// TwinCAT 3 PLC project PMPS_Prototype_Arbiter
// Title: PMPS
// Company: SLAC
// ProjectVersion: 0.0.0
// ProgramVersion: 3.1.4022.1
// libraries:
//   LCLS General, * (SLAC)
//   Tc2_MC2, * (Beckhoff Automation GmbH)
//   Tc2_Standard, * (Beckhoff Automation GmbH)
//   Tc2_System, * (Beckhoff Automation GmbH)
//   Tc2_Utilities, * (Beckhoff Automation GmbH)
//   Tc3_Database, * (Beckhoff Automation GmbH)
//   Tc3_EventLogger, * (Beckhoff Automation GmbH)
//   Tc3_Module, * (Beckhoff Automation GmbH)
//   VisuDialogs, * (System)
//   TcUnit,newest,www.tcunit.org
//   VisuSymbols,3.5.10.0,System
// project tree:
//   DUTs/ E_ExampleDeviceStates.TcDUT, ST_BinarySolidAttenuator.TcDUT, ST_Device.TcDUT, ST_DeviceState.TcDUT (not stored), ST_DeviceStateExt.TcDUT (not stored), ST_DeviceStateTable.TcDUT, ST_SolidAttenuatorBlade.TcDUT (not stored)
//   / GlobalTextList.TcGTLO, ImagePool.TcIPO (not stored), PlcTask.TcTTO, Visualization Manager.TcVMO (not stored), VISU_TASK.TcTTO
//   GVLs/ GVL.TcGVL, PMPS_GVL_BeamParams.TcGVL
//   pmps-lib/HelperFunctions/ F_DeviceState_To_DeviceStateExt.TcPOU, F_DiffBeamParamsRB.TcPOU, F_DifferentBeamParams.TcPOU, F_DiffReqBeamParams.TcPOU, F_eVRangeCalculator.TcPOU, F_eVWithinSpec.TcPOU, F_SafeBPCompare.TcPOU (not stored), F_SetBeamParams.TcPOU, F_SetStateParams.TcPOU
//   pmps-lib/MajorComponents/ BeamParameterTransitionManager.TcPOU, FB_Arbiter.TcPOU, FB_BeamClassOutputs.TcPOU, FB_BeamParamAssertionPool.TcPOU, FB_BeamParamFanout.TcPOU, FB_BPRequestor.TcPOU, FB_FastFault.TcPOU, FB_HardwareFFOutput.TcPOU, FB_LinearDeviceStateTable.TcPOU, FB_LinearGovernor.TcPOU, FB_PhotonEnergyWatcher.TcPOU, FB_UsualSuspects.TcPOU
//   pmps-lib/TestComponents/ eBPTMTestStates.TcDUT, FB_Arbiter_Test.TcPOU, FB_AttenuatorSimulator.TcPOU, FB_BeamParamFanout_Test.TcPOU (excluded from build), FB_BPRequestor_Test.TcPOU (excluded from build), FB_BPTM_Test.TcPOU, FB_evRangeCalculator_Test.TcPOU, FB_eVWithinSpec_Test.TcPOU, FB_FastFault_Test.TcPOU, FB_MachineSimulator.TcPOU, FB_PhotonEnergyWatcher_Test.TcPOU, FB_SafeBPCompare_Test.TcPOU, FB_SolidAttenuator.TcPOU
//   POUs/DatabaseComponents/ FB_ExampleDeviceSM_DB.TcPOU, FB_MySQL_Client.TcPOU, F_DB_To_hTable.TcPOU
//   POUs/DeviceImplementationEx1/ FB_ExampleDevice.TcPOU (not stored), FB_ExampleDeviceSM.TcPOU
//   POUs/DeviceImplementationEx2/ FB_ExampleDeviceSM_All.TcPOU
//   POUs/ Fast_Faults_Setup.TcPOU, Fast_Faults_Evaluate.TcPOU, MachineSimulation.TcPOU, MAIN.TcPOU, PMPS_Arbiter.TcPOU, TestSetups.TcPOU
//   Version/ Global_Version.TcGVL
//   VISUs/ ArbiterStats.TcVIS, BeamParameterStats.TcVIS, FastFaultGUI.TcVIS, ImagerGUI.TcVIS, PhotonEnergyWatcher.TcVIS, Visualization.TcVIS, WordBitDisplay.TcVIS
// real-time tasks:
//   TASK PlcTask: cycle T#1ms, priority 20, ADS port 350
//   TASK VISU_TASK: cycle T#200000us, priority 30, ADS port 351
//   TASK PlcTask1: cycle T#10ms, priority 21, ADS port 352
// motion (NC):
//   TASK NC-Task 1 SAF: cycle T#2ms, priority 4, ADS port 501
//   TASK NC-Task 1 SVB: cycle T#10ms, priority 8, ADS port 511
//   AXIS Dev1 (id 1)
//   AXIS Dev 2 (id 2)
//   AXIS Axis 3 (id 3)
// I/O:
//   DEVICE Device 1 (EtherCAT) (disabled), AmsNetId 169.254.224.1.2.1
//     Term 1 (EK1200) [EK1200-5000 EtherCAT Power supply (2A E-Bus)]
//       Term 2 (EL2022) [EL2022 2Ch. Dig. Output 24V, 2A]
//       Term 10 (EL7047)
//       Term 3 (EK1122) [EK1122 2 port EtherCAT junction]
//         Box 8 (EL6692) [EL6692 EtherCAT Bridge terminal (Secondary)]
//         Box 9 (EL6692) [EL6692 EtherCAT Bridge terminal (Secondary)]
//       Term 4 (EK1110) [EK1110 EtherCAT extension]
//   DEVICE Device 2 (EtherCAT) (disabled), AmsNetId 169.254.224.1.3.1
//     Term 1 (EK1200) [EK1200-5000 EtherCAT Power supply (2A E-Bus)]
//       Term 6 (EL6692) [EL6692 EtherCAT Bridge terminal (Primary)]
//       Term 3 (EL9011) [EL9011 End Terminal]
// variable links:
//   PMPS_Prototype_Arbiter Instance <-> Device 1 (EtherCAT)/Term 1 (EK1200)/Term 3 (EK1122)/Box 8 (EL6692)
//     PlcTask Inputs/MachineSimulation.i_SimReqBP <-> IO Inputs/RequestBP
//     PlcTask Outputs/MachineSimulation.q_SimCurrBP <-> IO Outputs/CurrentBP
//   PMPS_Prototype_Arbiter Instance <-> NC-Task 1 SAF/Axes/Dev 2
//     PlcTask Inputs/MAIN.fbDev2.stDevice.stAxis.NcToPlc <-> Outputs/ToPlc
//     PlcTask Outputs/MAIN.fbDev2.stDevice.stAxis.PlcToNc <-> Inputs/FromPlc
//   PMPS_Prototype_Arbiter Instance <-> NC-Task 1 SAF/Axes/Dev1
//     PlcTask Inputs/MAIN.fbDev1.stDevice.stAxis.NcToPlc <-> Outputs/ToPlc
//     PlcTask Outputs/MAIN.fbDev1.stDevice.stAxis.PlcToNc <-> Inputs/FromPlc

CONFIGURATION PMPS_Prototype_Arbiter
    RESOURCE PLC ON TwinCAT3
        TASK PlcTask(INTERVAL := T#1ms, PRIORITY := 20);
        TASK VISU_TASK(INTERVAL := T#200000us, PRIORITY := 30);
        PROGRAM MAIN WITH PlcTask : MAIN;
        PROGRAM VisuElems_Visu_Prg WITH VISU_TASK : VisuElems.Visu_Prg;
    END_RESOURCE
END_CONFIGURATION

// ---- DUTs/E_ExampleDeviceStates.TcDUT
{attribute 'qualified_only'}
{attribute 'strict'}
TYPE E_ExampleDeviceStates :
(
	enum_member := 0
);
END_TYPE

// ---- DUTs/ST_BinarySolidAttenuator.TcDUT
TYPE ST_BinarySolidAttenuator :
STRUCT
	axBlades	: ARRAY [0..9] OF ST_SolidAttenuatorBlade;
END_STRUCT
END_TYPE

// ---- DUTs/ST_Device.TcDUT
TYPE ST_Device :
STRUCT
	//IO
	stAxis	:	AXIS_REF;
	//The following limit switches must be TRUE or high (ie. NC) to enable that direction of motion
	//The EPICS display should show an inverted indicator to communicate end of travel reached
	i_xLoLim	AT %I*	:	BOOL; //Wire normally-closed
	i_xHiLim	AT %I*	:	BOOL; //Wire normally-closed
	
	//Acuator Parameters
	lrUpperPositionLimit	:	LREAL := 10000000000; //Use in conjuntion with limit switches or set to a huge number to ignore
	lrLowerPositionLimit	:	LREAL := -10000000000; //Use in conjuntion with limit switches or set to a huge number to ignore
	
	xEnable	:	BOOL := TRUE;
	
	//Supervisory System
	
	//MPS Override
	xOverrideMPSLimits	: BOOL := FALSE; //Set true to move beyond MPS limits. Note this will trip beam off.
	
	//Device States
	StateTable		:	FB_LinearDeviceStateTable;
	
	stTransitionState	:	ST_DeviceState; //The transition state might have non-zero beam parameters
	nSafeState			:	UDINT; //State where the device is considered safe
	nTransitionState	:	UDINT;
	
	nRequestedState	:	UDINT; //EPICS control, cleaned (checked against array limits) and deposited in nTargetState
	nTargetState	:	UDINT; //The requested state should be deposited here after cleaning
	nActiveState	:	UDINT; //The last successfully reached state
	
	
END_STRUCT
END_TYPE

// ---- DUTs/ST_DeviceStateTable.TcDUT
TYPE ST_DeviceStateTable :
STRUCT
	iDeviceID:DINT;
	iStateID:DINT;
	rTargetPosition: REAL;
	rTolerance: REAL;
	rTransmission: REAL;
	iBeamClass : DINT;
	rPhotonEnergy: REAL;
END_STRUCT
END_TYPE

// ---- pmps-lib/TestComponents/eBPTMTestStates.TcDUT
{attribute 'qualified_only'}
{attribute 'strict'}
TYPE eBPTMTestStates :
(
	Init := 0,
	WaitingForValidID := 50,
	WaitingForTransitionAssertion := 100,
	WaitingForFinalAssertion	:= 200,
	Transitioning	:= 300,
	CleaningUp	:= 400,
	AnotherState := 500
);
END_TYPE

// ---- GVLs/GVL.TcGVL

VAR_GLOBAL
	g_fbArbiter1	:	FB_Arbiter;
	g_fbArbiter2	:	FB_Arbiter;
	{attribute 'TcLinkTo' := '.q_xFastFaultOut:=TIIB[PMPS_FFO]^Channel 1^Output'}
	g_FastFaultOutput1	:	FB_HardwareFFOutput;
	g_rTestingVelocity	:	LREAL := VISIBLE_TEST_VELOCITY;
	g_fbFFRegistry	:	FB_UsualSuspects;
END_VAR

VAR_GLOBAL CONSTANT
	EXCLUDED_ASSERTION_ID	:	UDINT	:= 16#FFFFFFFF; //An assertion ID that should always return "not found" in the assertion pool
	VISIBLE_TEST_VELOCITY	:	LREAL	:= 10;
	FAST_TEST_VELOCITY		:	LREAL	:= 100;
	MAX_DEVICE_STATES		:	UDINT	:= 300;
END_VAR

// ---- GVLs/PMPS_GVL_BeamParams.TcGVL
{attribute 'qualified_only'}
VAR_GLOBAL
	stReqFBDBeamParamsSum	:	ST_BeamParams;
	stReqMethBeamParamSum	:	ST_BeamParams;
	stCurrentBeamParameters	:	ST_BeamParams;
END_VAR
VAR_GLOBAL CONSTANT
	cstFullBeam	:	ST_BeamParams := (
		fAtt := 0,
		fPP_mJ := 1E4,
		neVRange := 2#1111_1111_1111_1111,
		nRate	:= UDINT#1000000
		
);
	cstSafeBeam	:	ST_BeamParams := (
		fAtt := 100,
		fPP_mJ := 0,
		neVRange := 0,
		nRate	:= 0
);
	cnMaxStateArrayLen : INT := 20;
	
	MAX_ASSERIONS	:	UDINT := 100; //Maximum number of assertions permitted in the arbiter
	
	g_cBoundaries	:	INT	:= 15;
	g_areVBoundaries	:	ARRAY [0..g_cBoundaries]	OF	REAL	:= [
	0.2,
	0.3,
	0.4,
	0.5,
	0.6,
	0.7,
	0.8,
	0.9,
	1.0,
	1.1,
	1.2,
	1.3,
	1.4,
	1.5,
	1.6,
	1.7
];
END_VAR

// ---- Version/Global_Version.TcGVL
{attribute 'TcGenerated'}
// This function has been automatically generated from the project information.
VAR_GLOBAL CONSTANT
	{attribute 'const_non_replaced'}
	{attribute 'linkalways'}
	stLibVersion_PMPS : ST_LibVersion := (iMajor := 0, iMinor := 0, iBuild := 0, iRevision := 0, sVersion := '0.0.0');
END_VAR

// ---- POUs/MAIN.TcPOU
PROGRAM MAIN
VAR
	fbDev1	:	FB_ExampleDeviceSM_All;
	fbDev2	:	FB_ExampleDeviceSM_All;
	
	rtInit	:	R_TRIG;
	Initialize	:	BOOL := TRUE;
	
	DemoMode: BOOL :=FALSE;
	//fbDev3	:	FB_ExampleDeviceSM_DB;

END_VAR

//Sub-system Device PLC

IF DemoMode	THEN

//Fast Faults must run first
Fast_Faults_Setup();

IF Initialize THEN
	fbDev1(cBase := 10,
		fbFastFaultOutput := g_FastFaultOutput1,
		fbArbiter := g_fbArbiter1);
	fbDev2(cBase := 1000,
		fbFastFaultOutput := g_FastFaultOutput1,
		fbArbiter := g_fbArbiter1);
	g_fbArbiter1.A_Init();

//	fbDev3(cBase := 0,iDBID:=1,sDBNetId:='172.21.42.53.1.1',sDeviceID:='1',
//		fbArbiter := g_fbArbiter,
//		fbFastFaultOutput := g_FastFaultOutput1);
	Initialize := FALSE;
END_IF

//Example devices
fbDev1(fbFastFaultOutput := g_FastFaultOutput1,
		fbArbiter := g_fbArbiter1);
fbDev2(fbFastFaultOutput := g_FastFaultOutput1,
		fbArbiter := g_fbArbiter1);


//fbDev3(fbArbiter := g_fbArbiter,
//		fbFastFaultOutput := g_FastFaultOutput1);
		

		
PMPS_Arbiter();

Fast_Faults_Evaluate();

MachineSimulation();

ELSE
	TestSetups();
END_IF

ACTION FB_Vis:
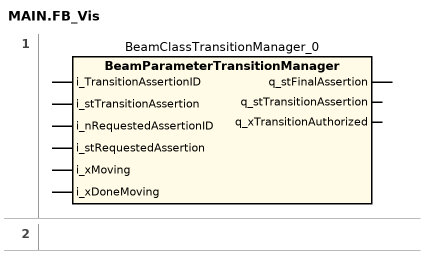
// NETWORK 1
BeamClassTransitionManager_0(); // BeamParameterTransitionManager

// NETWORK 2
END_ACTION

ACTION Initialize:

END_ACTION

END_PROGRAM

// ---- POUs/DeviceImplementationEx2/FB_ExampleDeviceSM_All.TcPOU
(* This version of the block is self contained. Minimizes wiring.*)
FUNCTION_BLOCK FB_ExampleDeviceSM_All
VAR_INPUT
	cBase: UDINT;
END_VAR
VAR_OUTPUT
END_VAR
VAR_IN_OUT
	fbFastFaultOutput	:	FB_HardwareFFOutput;
	fbArbiter	:	FB_Arbiter;
END_VAR
VAR
	stDevice	:	ST_Device;
	fbGovernor	:	FB_LinearGovernor;
	mcPower	:	MC_Power;
	mcStop: MC_Stop;
	mcAbsolute	:	MC_MoveAbsolute;
	fbBPTM	:	BeamParameterTransitionManager;
	xStartMove: BOOL;
	
	stCheckState: ST_DeviceState;
	stTargetState	:	ST_DeviceState; //Target device state

END_VAR
VAR PERSISTENT
	nLastActiveState	:	UDINT;
END_VAR

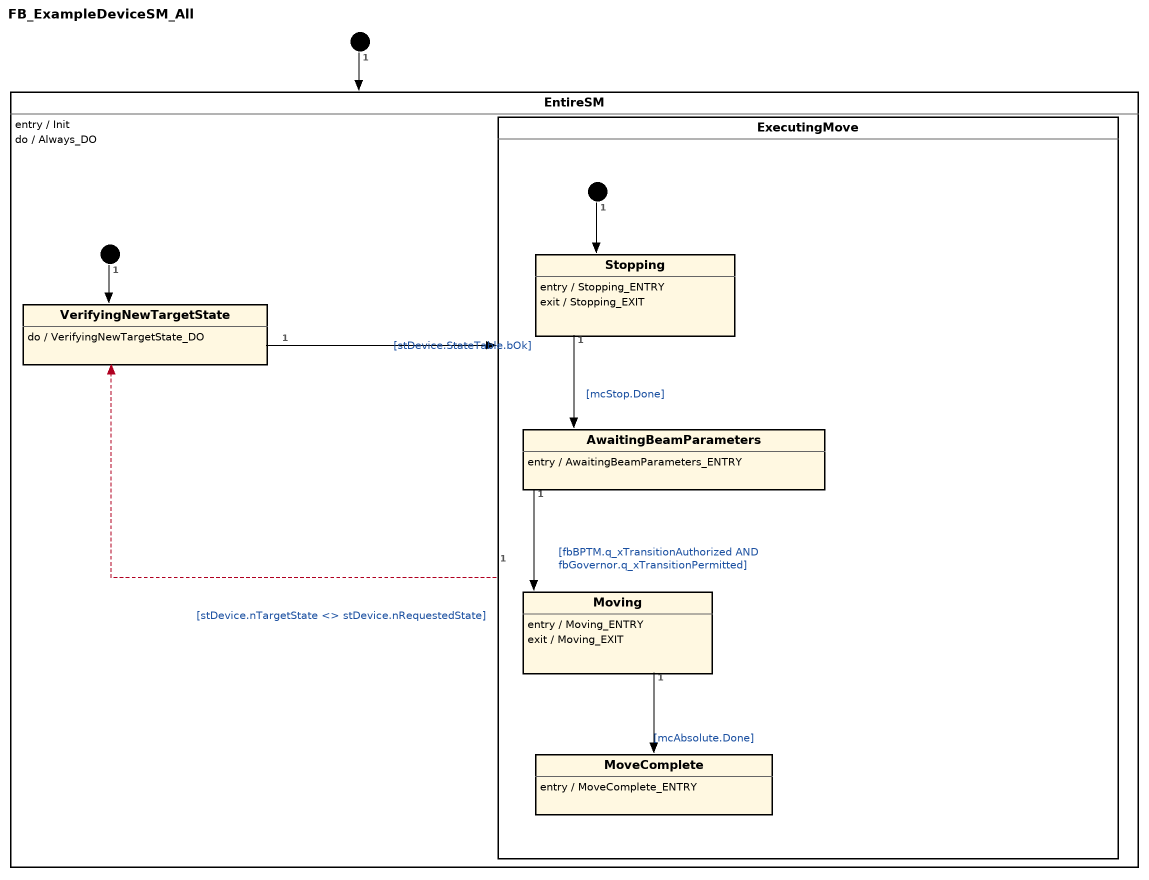
STATECHART FB_ExampleDeviceSM_All  // abortable
    START StartState3
    COMPOSITE STATE EntireSM
        entry / Init
        do / Always_DO
        START StartState1
        COMPOSITE STATE ExecutingMove
            START StartState2
            STATE Stopping
                entry / Stopping_ENTRY
                exit / Stopping_EXIT
            STATE AwaitingBeamParameters
                entry / AwaitingBeamParameters_ENTRY
            STATE Moving
                entry / Moving_ENTRY
                exit / Moving_EXIT
            STATE MoveComplete
                entry / MoveComplete_ENTRY
            StartState2 -> Stopping  // priority 1, on completion
            Stopping -> AwaitingBeamParameters [mcStop.Done] // priority 1, rising edge
            AwaitingBeamParameters -> Moving [fbBPTM.q_xTransitionAuthorized AND fbGovernor.q_xTransitionPermitted] // priority 1, rising edge
            Moving -> MoveComplete [mcAbsolute.Done] // priority 1, rising edge
        END_STATE
        STATE VerifyingNewTargetState
            do / VerifyingNewTargetState_DO
        StartState1 -> VerifyingNewTargetState  // priority 1, on completion
        ExecutingMove -> VerifyingNewTargetState [stDevice.nTargetState <> stDevice.nRequestedState] // priority 1, exception, rising edge
        VerifyingNewTargetState -> ExecutingMove [stDevice.StateTable.bOk] // priority 1
    END_STATE
    StartState3 -> EntireSM  // priority 1, on completion
END_STATECHART

ACTION Always_DO:
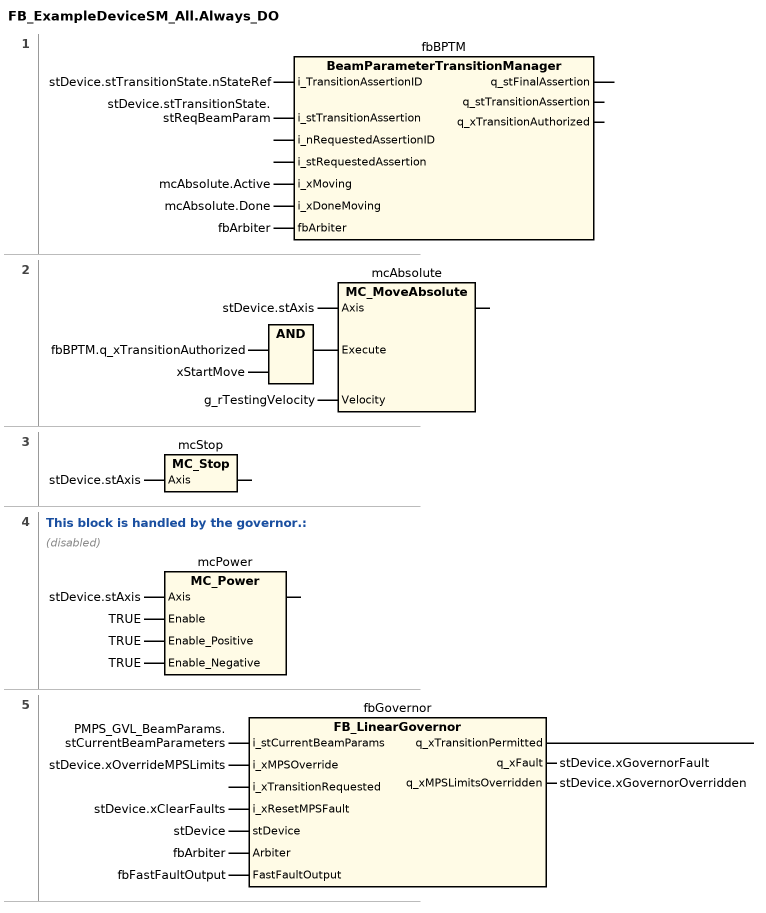
// NETWORK 1
fbBPTM(
    i_TransitionAssertionID := stDevice.stTransitionState.nStateRef,
    i_stTransitionAssertion := stDevice.stTransitionState.stReqBeamParam,
    i_xMoving := mcAbsolute.Active,
    i_xDoneMoving := mcAbsolute.Done,
    fbArbiter := fbArbiter); // BeamParameterTransitionManager

// NETWORK 2
mcAbsolute(
    Axis := stDevice.stAxis,
    Execute := fbBPTM.q_xTransitionAuthorized AND xStartMove,
    Velocity := g_rTestingVelocity); // MC_MoveAbsolute

// NETWORK 3
mcStop(Axis := stDevice.stAxis); // MC_Stop

// NETWORK 4 (disabled)
// label: This block is handled by the governor.
// mcPower(Axis := stDevice.stAxis, Enable := TRUE, Enable_Positive := TRUE, Enable_Negative := TRUE); // MC_Power

// NETWORK 5
fbGovernor(
    i_stCurrentBeamParams := PMPS_GVL_BeamParams.stCurrentBeamParameters,
    i_xMPSOverride := stDevice.xOverrideMPSLimits,
    i_xResetMPSFault := stDevice.xClearFaults,
    stDevice := stDevice,
    Arbiter := fbArbiter,
    FastFaultOutput := fbFastFaultOutput,
    q_xFault => stDevice.xGovernorFault,
    q_xMPSLimitsOverridden => stDevice.xGovernorOverridden); // FB_LinearGovernor
END_ACTION

ACTION AwaitingBeamParameters_ENTRY:
fbBPTM.i_stRequestedAssertion := stTargetState.stReqBeamParam;
fbBPTM.i_nRequestedAssertionID := stTargetState.nStateRef;

//Tell the governor that we're trying to move.
fbGovernor.i_xTransitionRequested := TRUE;
END_ACTION

ACTION Init:

//Safe State
stDevice.nSafeState := cBase;
stDevice.nTransitionState := cBase+100;

//Initialize the State Table
stDevice.StateTable.A_Reset();

//Device State Table Instantiation
//To be done by the device state table database system
F_SetStateParams(
	nStateRef := stDevice.nSafeState,
	rPosition := 0,
	rTolerance := 10,
	stBeamParams := PMPS_GVL_BeamParams.cstFullBeam,
	Table := stDevice.StateTable
);
F_SetStateParams(
	nStateRef := cBase + 1,
	rPosition := 100,
	rTolerance := 10,
	stBeamParams := F_SetBeamParams(
		fAtt := 20,
		fPP_mJ := 1,
		neVReqRange	:= 2#1111_1011_1111_0000,
		nRate := 10
		),
	Table := stDevice.StateTable
);
F_SetStateParams(
	nStateRef := cBase + 2,
	rPosition := 200,
	rTolerance := 10,
	stBeamParams := F_SetBeamParams(
		fAtt := 30,
		fPP_mJ := 1,
		neVReqRange	:= 2#1111_1011_1111_0000,
		nRate := 10
		),
	Table := stDevice.StateTable
);
F_SetStateParams(
	nStateRef := cBase + 3,
	rPosition := 300,
	rTolerance := 10,
	stBeamParams := F_SetBeamParams(
		fAtt := 20,
		fPP_mJ := 1,
		neVReqRange	:= 2#1111_1011_1111_0000,
		nRate := 10
		),
	Table := stDevice.StateTable
);

F_SetStateParams(
	nStateRef := stDevice.nTransitionState,
	rPosition := 0,
	rTolerance := 0,
	stBeamParams := F_SetBeamParams(
		fAtt := 0,
		fPP_mJ := 0,
		neVReqRange	:= 2#1111_1011_1111_0000,
		nRate := 0
		),
	Table := stDevice.StateTable
);

//Set device transition state
stDevice.StateTable.A_Lookup(
	key := stDevice.nTransitionState,
	getValue => stDevice.stTransitionState
);

//Need an initialization routine for setting the active state
//Check if the device is at safe state
//If the device is within the state boundaries, it's considered to be in that state
stDevice.StateTable.A_Lookup(key:= stDevice.nSafeState);
IF stDevice.StateTable.bOk THEN
	stCheckState := stDevice.StateTable.getValue;
ELSE
	stCheckState := stDevice.stTransitionState; //This needs to be safer <TODO>
END_IF

IF stDevice.stAxis.NcToPlc.ActPos <= stCheckstate.rPosition + stCheckState.rTolerance AND
	stDevice.stAxis.NcToPlc.ActPos >= stCheckState.rPosition - stCheckState.rTolerance THEN
	stDevice.nActiveState := nLastActiveState;
ELSE
	stDevice.nActiveState := stDevice.nTransitionState;
END_IF

//Simulation Hardware Limit Switches
stDevice.i_xHiLim := TRUE;
stDevice.i_xLoLim := TRUE;
END_ACTION

ACTION MoveComplete_ENTRY:
//Clear transition request
fbGovernor.i_xTransitionRequested := FALSE;
//Latch active state
stDevice.nActiveState := stDevice.nTargetState;
nLastActiveState := stDevice.nActiveState;
END_ACTION

ACTION Moving_ENTRY:
xStartMove := TRUE;
mcAbsolute.Position := stTargetState.rPosition;
END_ACTION

ACTION Moving_EXIT:
xStartMove := FALSE;
END_ACTION

ACTION NewMove_ENTRY:

END_ACTION

ACTION Stopping_ENTRY:
mcStop.Execute := TRUE;
END_ACTION

ACTION Stopping_EXIT:
mcStop.Execute := FALSE;
END_ACTION

ACTION VerifyingNewTargetState_DO:
stDevice.StateTable.A_Lookup(
	key := stDevice.nRequestedState
);

IF stDevice.StateTable.bOk THEN
	stTargetState := stDevice.StateTable.getValue;
	stDevice.nTargetState := stDevice.nRequestedState;
ELSE
	; //log ignored state/ generate an error? <TODO>
END_IF
END_ACTION

END_FUNCTION_BLOCK

// ---- pmps-lib/MajorComponents/FB_HardwareFFOutput.TcPOU

FUNCTION_BLOCK FB_HardwareFFOutput
VAR_INPUT
	i_xReset	:	BOOL;
	i_xVeto	:	BOOL;	
END_VAR
VAR_OUTPUT
	q_xFastFaultOut	AT %Q*	:	BOOL;
END_VAR
VAR
	xOK	:	BOOL;
	rtReset	:	R_TRIG;
	
	//Fault registration list
	//Fast faults add their name here to indicate they
	//"check in" to indicate their status with this fast
	//fault output. ie. They may be a culprit of beam off.
	asList	:	ARRAY[0..99] OF T_MaxString;
	nIndex	:	INT;
END_VAR
VAR CONSTANT
	cMaxList	:	INT := 99;
END_VAR

rtReset(CLK:=i_xReset);
xOK S= rtReset.Q;
// <TODO> latch off beam if DI card status goes bad

METHOD CheckIn : BOOL
VAR_INPUT
	i_xOK	:	BOOL; //Keep true to keep beam
END_VAR
IF NOT i_xOK THEN
	THIS^.xOK := FALSE; //Very clever, thanks Zach!
END_IF
END_METHOD

ACTION EvaluateOutput:
//<TODO> add diagnostic for success or failure of reset
q_xFastFaultOut := xOK OR i_xVeto;
END_ACTION

METHOD Register : BOOL
VAR_INPUT
	i_sFFName	:	STRING; //Fast fault FB variable name to register
END_VAR

VAR
END_VAR
IF THIS^.nIndex <= THIS^.cMaxList THEN
	THIS^.asList[MIN(THIS^.nIndex,THIS^.cMaxList)]:=i_sFFName;
	THIS^.nIndex := THIS^.nIndex + 1;
	Register := TRUE; //Add successful
ELSE
	Register := FALSE; //failed to add name to list
END_IF
END_METHOD

END_FUNCTION_BLOCK

// ---- pmps-lib/MajorComponents/FB_Arbiter.TcPOU
(* FB Arbiter

The arbiter primary objectives are:
- Provide a simple interface for devices to request beam parameter sets
- Provide a way for devices to verify their BPS is active in the arbiter
- Provide a way for devices remove their requests from evaluation
- Evaluate all active beam parameter requests registered with the aribiter,
to determine the safest combination of all sets, provide this set as an output.
- Do all of this with minimal overhead

To these ends, the arbiter uses a hash-table, the rows being a state-id as the key, and a corresponding
 beam parameter set to be evaluated against all the other sets (or rows), in the table.
 
The hash table can be thought of as an array on steriods, they are worth reading about, suffice to say
the hash table will tell you when you reach the end of all the entries, and enables us to find entries quickly.

These features efficiently address the addition, removal, and verification of beam parameter sets listed in the above requirements.

An important thing to pay attention to is the A_Arbitrate action. This action implements the evaluation of beam parameter
sets against each other.

*)

FUNCTION_BLOCK FB_Arbiter
VAR_INPUT
	i_nStateID	:	UDINT; //Set to the stateID of the state requesting the beam parameter set
	i_stAssertBeamParams	:	ST_BeamParams; //Set to the beam parameter set of the state required
END_VAR
VAR_OUTPUT
	q_stBeamParams	:	ST_BeamParams; //Updated on each cycle of the arbiter FB with the current arbitrated beam parameter set
	
	q_xStateIDFound	:	BOOL; //Set true if a state-id is found in the assertion pool after calling A_VerifyAssertion
END_VAR
VAR
	
	fbBPAssertionPool	:	FB_BeamParamAssertionPool; //Table of active beam parameter assertions
	
	getPosPtr	: POINTER TO T_HashTableEntry := 0; 
	getBPStruct	:	ST_BeamParams;
	stOutputBP	:	ST_BeamParams; //Safest beam parameters from all in the assertion pool
	
	
END_VAR

ACTION A_Init:
// Clears the entire beam parameter assertion pool (hashtable).

fbBPAssertionPool.A_Reset();
END_ACTION

METHOD AddRequest : BOOL
VAR_INPUT
	nReqID	:	DWORD; //StateID of state requesting beam parameter set
	stReqBP		:	ST_BeamParams; //Requested beam params
END_VAR
IF THIS^.CheckRequest(nReqID) THEN
	AddRequest := FALSE;
	RETURN;
END_IF

IF nReqID <> EXCLUDED_ASSERTION_ID THEN
	THIS^.fbBPAssertionPool.A_Add(
		key := nReqID,
		putValue := stReqBP
	);
END_IF
	
IF NOT THIS^.fbBPAssertionPool.bOk THEN
	; //Overflow <TODO>
END_IF

AddRequest := THIS^.fbBPAssertionPool.bOk;
END_METHOD

METHOD ArbitrateBP : ST_BeamParams
VAR_INPUT
	stBP1	:	ST_BeamParams;
	stBP2	:	ST_BeamParams;
END_VAR
//<TODO>Add something here to register the key that won for each param

//Attenuation
ArbitrateBP.fAtt := MAX(stBP1.fAtt, stBP2.fAtt);

//Pulse energy
ArbitrateBP.fPP_mJ := MIN(stBP1.fPP_mJ, stBP2.fPP_mJ);

//Photon energy ranges
ArbitrateBP.neVRange := stBP1.neVRange AND stBP2.neVRange;

//Rate
ArbitrateBP.nRate := MIN(stBP1.nRate, stBP2.nRate);
END_METHOD

(* Searches state assertion pool for a state-id, and sets q_xStateIDFound true if found.

Use like so:

fbArbiter.A_VerifyAssertion(
i_nStateId := nStateIDAssertionToCheck
);

IF fbArbiter.q_xStateIDFound THEN:
	Do something
ELSE:
	Don't do something

*)
METHOD CheckRequest : BOOL
VAR_INPUT
	nReqID	:	DWORD;
END_VAR
THIS^.fbBPAssertionPool.A_Lookup(key := nReqID);

CheckRequest := THIS^.fbBPAssertionPool.bOk;
END_METHOD

METHOD GetArbitratedBP : ST_BeamParams
VAR_INPUT
END_VAR
VAR
	getPosPtr	: POINTER TO T_HashTableEntry := 0;
	getBPStruct	:	ST_BeamParams;
	
	stOutputBP	:	ST_BeamParams; //Holding struct for arbitration process
END_VAR
//Arbitrate
(*
This step cycles through every hash table entry, comparing
the beam parameters from each assertion to what we're planning
to assert.

The safer of the two parameters is kept so at the end we may
have a mix of beam parameters, the composition being safe for
all asserters.

*)

THIS^.fbBPAssertionPool.A_GetFirst( putPosPtr := 0, getPosPtr=>getPosPtr, getValue=>getBPStruct );
IF THIS^.fbBPAssertionPool.bOk THEN //If the table is empty (not OK), we are left with the default stOutputBP set above.
	
	//The first entry in the hash table is taken as the setting to arbitrate against
	stOutputBP := F_SetBeamParams(
		fAtt := getBPStruct.fAtt,
		fPP_mJ := getBPStruct.fPP_mJ,
		neVRange	:= getBPStruct.neVRange,
		nRate := getBPStruct.nRate
	);

	REPEAT
		THIS^.fbBPAssertionPool.A_GetNext( putPosPtr := THIS^.fbBPAssertionPool.getPosPtr, getPosPtr=>getPosPtr, getValue=>getBPStruct );
		IF THIS^.fbBPAssertionPool.bOk THEN
			stOutputBP := ArbitrateBP(stOutputBP, getBPStruct);
		END_IF
	UNTIL NOT fbBPAssertionPool.bOk
	END_REPEAT
ELSE
	//Safest parameters to start
	stOutputBP := PMPS_GVL_BeamParams.cstSafeBeam;
END_IF

THIS^.q_stBeamParams := stOutputBP;

GetArbitratedBP.fAtt := stOutputBP.fAtt;
GetArbitratedBP.fPP_mJ := stOutputBP.fPP_mJ;
GetArbitratedBP.nBeamClass := stOutputBP.nBeamClass;
GetArbitratedBP.neVRange := stOutputBP.neVRange;
GetArbitratedBP.nRate := stOutputBP.nRate;
GetArbitratedBP.xValidToggle := NOT GetArbitratedBP.xValidToggle;
END_METHOD

(* Searches for a state-id, and removes it from the assertion pool.

Use like so:
fbArbiter.A_RemoveAssertion(
i_nStateId := nStateIDAssertionToRemove
);

*)
METHOD RemoveRequest : BOOL
VAR_INPUT
	nReqId	:	DWORD;
END_VAR
IF nReqId <> EXCLUDED_ASSERTION_ID THEN
	THIS^.fbBPAssertionPool.A_Remove(key := nReqId);
	
	IF THIS^.fbBPAssertionPool.bOk THEN
		;
	ELSE
		;
	END_IF
END_IF

RemoveRequest := THIS^.fbBPAssertionPool.bOk;
END_METHOD

END_FUNCTION_BLOCK

// ---- pmps-lib/MajorComponents/FB_BeamParamAssertionPool.TcPOU
(* This function block implements simple database. Data element values are stored in the hash table.  *)
FUNCTION_BLOCK FB_BeamParamAssertionPool
VAR_INPUT
	key 		: DWORD := 0;(* Entry key: used by A_Lookup, A_Remove method, the key variable is also used by A_Add method *)
	putPosPtr	: POINTER TO T_HashTableEntry := 0;(* Hash table entry position pointer (used by A_Find, A_GetNext, A_GetPrev) *)
	putValue 	: ST_BeamParams;(* Hash table entry value (used by A_AddHead, A_AddTail, A_Find )*)
END_VAR
VAR_OUTPUT
	bOk			: BOOL := FALSE;(* TRUE = Success, FALSE = Failed *)
	getPosPtr	: POINTER TO T_HashTableEntry := 0;(* Returned hash table entry position pointer *)
	getValue 	: ST_BeamParams;(* Returned hash table entry value *)
	nCount		: UDINT := 0;(* Hash table size (number of used entries, used by A_Count) *)
END_VAR
VAR
	dataPool	: ARRAY[0..PMPS_GVL_BeamParams.MAX_ASSERIONS] OF ST_BeamParams;(* Structured data element pool *)
	entries		: ARRAY[0..PMPS_GVL_BeamParams.MAX_ASSERIONS] OF T_HashTableEntry;(* Max. number of hash table entries. The value of table entry = 32 bit integer (pointer to dataPool-array-entry) *)
	fbTable 	: FB_HashTableCtrl;(* basic hash table control function block *)
	hTable 		: T_HHASHTABLE;(* hash table handle *)
	pRefPtr		: POINTER TO ST_BeamParams := 0;
	indexOfElem	: ULINT;(* Integer value (max. size: x86=>32bit, x64=>64bit)*)
END_VAR

;

ACTION A_Add:
(* Adds entry to the table *)
MEMSET( ADR( getValue ), 0, SIZEOF( getValue ) );
getPosPtr := 0;

fbTable.A_Add( hTable := hTable, key := key, putValue := ADR(PMPS_GVL_BeamParams.cstSafeBeam)(* we will set this value later *), getPosPtr=>getPosPtr, bOk=>bOk );(* Add new element to the table, getPosPtr points to the new entry *)
IF fbTable.bOk THEN(* Success *)
	fbTable.A_GetIndexAtPosPtr( hTable := hTable, putPosPtr := getPosPtr, getValue =>indexOfElem, bOk=>bOk );(* Get array index of getPosPtr entry *)
	IF fbTable.bOk THEN(* Success *)
		pRefPtr 	:= ADR( dataPool[indexOfElem] );(* Get pointer to the data element *)

		pRefPtr^ := putValue;(* copy application value *)

		fbTable.A_Add( hTable := hTable, key := key, putValue := pRefPtr, bOk=>bOk );(* Assign the entry value = pointer to the data element *)
		IF fbTable.bOk THEN(* Success *)
			getValue := putValue;
		END_IF
	END_IF
END_IF
END_ACTION

ACTION A_Count:
(* Count number of used entries *)
nCount := hTable.nCount;
bOk := TRUE;
END_ACTION

ACTION A_GetFirst:
(* Get first entry position pointer and value *)
MEMSET( ADR( getValue ), 0, SIZEOF( getValue ) );
getPosPtr := 0;

fbTable.A_GetFirst( hTable := hTable, putPosPtr := putPosPtr, getValue=>pRefPtr, getPosPtr=>getPosPtr, bOk=>bOk );
IF fbTable.bOk THEN
	getValue := pRefPtr^;
END_IF
END_ACTION

ACTION A_GetNext:
(* Get next entry position pointer and value *)
MEMSET( ADR( getValue ), 0, SIZEOF( getValue ) );
getPosPtr := 0;
bOk := FALSE;

IF putPosPtr = 0 THEN
	RETURN;
END_IF

fbTable.A_GetNext( hTable := hTable, putPosPtr := putPosPtr, getValue=>pRefPtr, getPosPtr=>getPosPtr, bOk=>bOk );
IF fbTable.bOk THEN
	getValue := pRefPtr^;
END_IF
END_ACTION

ACTION A_Lookup:
(* Lookup for entry by key  *)
MEMSET( ADR( getValue ), 0, SIZEOF( getValue ) );
getPosPtr := 0;

fbTable.A_Lookup( key := key, hTable := hTable, putPosPtr := putPosPtr, getValue=>pRefPtr, getPosPtr=>getPosPtr, bOk=>bOk );
IF fbTable.bOk THEN
	getValue := pRefPtr^;
END_IF
END_ACTION

ACTION A_Remove:
(* Search for entry and remove it *)
MEMSET( ADR( getValue ), 0, SIZEOF( getValue ) );
getPosPtr := 0;

fbTable.A_Remove( key := key, hTable := hTable, putPosPtr := putPosPtr, getValue=>pRefPtr, getPosPtr=>getPosPtr, bOk=>bOk );
IF fbTable.bOk THEN
	getValue := pRefPtr^;
END_IF
END_ACTION

ACTION A_Reset:
(* Reset/initialize linked list *)
MEMSET( ADR( getValue ), 0, SIZEOF( getValue ) );
getPosPtr := 0;
bOk := F_CreateHashTableHnd( ADR( entries ), SIZEOF( entries ), hTable );(* Intialize table handle *)
fbTable.A_Reset( hTable := hTable, bOk=>bOk );
nCount := 0;
END_ACTION

END_FUNCTION_BLOCK

// ---- pmps-lib/HelperFunctions/F_SetBeamParams.TcPOU
FUNCTION F_SetBeamParams : ST_BeamParams
VAR_INPUT
	fAtt	:	REAL := 100;
	fPP_mJ: REAL := 0;
	neVRange	:	WORD := 0;
	nRate	:	UDINT := 0;
END_VAR
VAR
	BeamParams	:	ST_BeamParams;
	
END_VAR

BeamParams.fAtt := LIMIT(0,fAtt,100);
BeamParams.fPP_mJ := LIMIT(0,fPP_mJ,20);
BeamParams.neVRange := neVRange;
BeamParams.nRate	:= MIN(nRate,1000000);

F_SetBeamParams	:= BeamParams;

END_FUNCTION

// ---- pmps-lib/MajorComponents/FB_LinearGovernor.TcPOU

(* The governor is meant to check your work and keep you from making mistakes.

Checks:
Does your state match the device position and visa versa?
Are the beam parameters safe for the device state?
Did you properly assert the transition and final beam parameters?

*)
FUNCTION_BLOCK FB_LinearGovernor
VAR_INPUT
	i_stCurrentBeamParams	:	ST_BeamParams; //Link to global beam params
	i_xMPSOverride			:	BOOL; //True releases MPS limits after a delay
	i_xTransitionRequested	:	BOOL; //Set true to request a transition
	i_xResetMPSFault	:	BOOL; //Set true to clear MPS fault 
END_VAR
VAR_OUTPUT
	 //True when governor has released restrictions
	q_xTransitionPermitted	:	BOOL;
	//Set if MC_Power has an error, or override mode is requested
	q_xFault	:	BOOL; 
	// Indicates override mode is active
	q_xMPSLimitsOverridden: BOOL;
END_VAR
VAR_IN_OUT
	stDevice	:	ST_Device; //The governed
	Arbiter	:	FB_Arbiter;
	FastFaultOutput	:	FB_HardwareFFOutput;
END_VAR
VAR
	mcPower	:	MC_Power;
	
	xActuatorPositiveEnable: BOOL;
	xActuatorNegativeEnable: BOOL;
	
	xMPSPositiveEnable	:	BOOL;
	xMPSNegativeEnable	:	BOOL;
	lrPosition: LREAL;
	
	lrLatchedTargetPosition	:	LREAL;
	lrLatchedTargetTolerance	:	LREAL;
	stLatchedTargetState	:	ST_DeviceStateExt;
	
	lrMPSUpperLimit: LREAL;
	lrMPSLowerLimit: LREAL;
	rtNewState: R_TRIG;
	xTransitionOK: BOOL;
	
	tonMPSOverrideMode	:	TON := (
		PT := T#5S
	);
	
	srMPSFault	:	SR;
	// Actuator out of bounds fault
	xActuatorOOB: BOOL;
	//Beam parameters out of spec
	xBeamParamsOOS: BOOL;
	//Beam parameters of currently latched state
	
	stLatchedBeamParams: ST_BeamParams;
	stTargetState: ST_DeviceStateExt;
	
	rtLatchNewState	:	R_TRIG;
	xInit: BOOL := TRUE;
	
	stInitDeviceState: ST_DeviceStateExt;
	// Indicates an error with initialization
	xInitFault: BOOL;
	// Indicates the state could not be found in the state table. There may be something wrong in the device state machine implementation or state table instantiation.
	xStateLookupError: BOOL;
	// A transition needs to be requested at least once before we start latching any state.
	xTransitionHasBeenRequested: BOOL := FALSE;
	ffBeamParamsOK : FB_FastFault;
	ffActuatorBoundsOK	:	FB_FastFault;
END_VAR


lrPosition := stDevice.stAxis.NcToPlc.ActPos; //Actuator position

stDevice.stAxis.ReadStatus();
//Init
(* The init strategy is:
If the device is restored and it's residing at the safe position,
no PMPS faults. *)
////////////////////////////////
	IF xInit THEN
		xInit := FALSE;
		//Use nSafeSate for initialization. 
		stDevice.StateTable.A_Lookup(key := stDevice.nSafeState);
		IF stDevice.StateTable.bOk THEN
			stInitDeviceState := F_DeviceState_To_DeviceStateExt(stDevice.StateTable.getValue, TRUE);
			xInitFault := FALSE;
		ELSE
			xInitFault := TRUE;
			stInitDeviceState.xValid := FALSE;
		END_IF
		lrLatchedTargetPosition := stInitDeviceState.rPosition;
		lrLatchedTargetTolerance := stInitDeviceState.rTolerance;
		stLatchedBeamParams := stInitDeviceState.stReqBeamParam;
	END_IF

// The governor will permit transitions once it verifies the transition assertion is active
// Note the governor does not verify the target state beam params are asserted, perhaps it should <TODO>
////////////////////////////////
	IF i_xTransitionRequested THEN
		xTransitionHasBeenRequested	:= TRUE;
		
		xTransitionOK := Arbiter.CheckRequest( stDevice.stTransitionState.nStateRef) AND F_SafeBPCompare(i_stCurrentBeamParams, stDevice.stTransitionState.stReqBeamParam);
		
		//Set the target state for evaluation in further logic
		stdevice.StateTable.A_Lookup(key := stDevice.nTargetState);
		IF stDevice.StateTable.bOk THEN
			stTargetState := F_DeviceState_To_DeviceStateExt(stDevice.StateTable.getValue, TRUE);
			xStateLookupError := FALSE;
		ELSE
			xStateLookupError := TRUE;
			stTargetState.xValid := FALSE;
		END_IF
	ELSE
		xTransitionOK := FALSE;
	END_IF

(* Note about TransitionRequested

If TransitionRequested goes false during a transition, an MPS fault may be induced. This occurs
because the Actuator Out of Bounds fault will go back to using the original state limits, which
the axis may have already moved beyond.

To avoid this transient fault, make sure your device state machine is implemented such that the 
transition request to the governor block remains high until the target position is reached.
*)

//Determine if a transition is complete and latch the new state
(* A transition is complete when:

Axis at standstill.
Axis within tolerance.
No transition req.

Once these conditions are met, the MPS limits shall re-engage to restrict the
axis motion to the tolerance around the state position and the MPS fault monitors
shall evaluate based on the newly latched target state.
*)

rtLatchNewState(CLK := stDevice.stAxis.Status.StandStill AND
	lrPosition <= stTargetState.rPosition + stTargetState.rTolerance AND
	lrPosition >= stTargetState.rPosition - stTargetState.rTolerance AND
	NOT i_xTransitionRequested AND xTransitionHasBeenRequested);
	
IF rtLatchNewState.Q THEN
	lrLatchedTargetPosition := stTargetState.rPosition;
	lrLatchedTargetTolerance := stTargetState.rTolerance;
	stLatchedBeamParams := stTargetState.stReqBeamParam;
	stLatchedTargetState := stTargetState;
END_IF

//Let other blocks know the governor won't interfer with transitions
q_xTransitionPermitted := xTransitionOK;

//Adjust limit ranges based on active state and current target
IF xTransitionOK THEN
	//Extend range to include target state
	lrMPSUpperLimit := MAX(lrMPSUpperLimit, stTargetState.rPosition + stTargetState.rTolerance);
	lrMPSLowerLimit := MIN(lrMPSLowerLimit, stTargetState.rPosition - stTargetState.rTolerance);
ELSE
	//Calculate the limit positions for MPS based on current state
	lrMPSUpperLimit := lrLatchedTargetPosition + lrLatchedTargetTolerance;
	lrMPSLowerLimit := lrLatchedTargetPosition - lrLatchedTargetTolerance;
END_IF


//MPS override
(* In override mode, the device will be free to move anywhere within it's travel range *)
//Permit motion after a small delay
tonMPSOverrideMode(IN:=i_xMPSOverride OR stDevice.xOverrideMPSLimits, Q=>q_xMPSLimitsOverridden);

//Virtual limit switch evaluation
xActuatorPositiveEnable	:= stDevice.i_xHiLim AND lrPosition <= stDevice.lrUpperPositionLimit;
xActuatorNegativeEnable	:= stDevice.i_xLoLim AND lrPosition >= stDevice.lrLowerPositionLimit;

//Evaluate MPS limit states
xMPSPositiveEnable := lrPosition <= lrMPSUpperLimit;
xMPSNegativeEnable := lrPosition >= lrMPSLowerLimit;

//Final Limit switch evaluation
mcPower.Enable_Positive := xActuatorPositiveEnable AND (tonMPSOverrideMode.Q OR xMPSPositiveEnable);
mcPower.Enable_Negative := xActuatorNegativeEnable AND (tonMPSOverrideMode.Q OR xMPSNegativeEnable);

mcPower(
	Axis := stDevice.stAxis,
	Enable := stDevice.xEnable //link to device enable <TODO>
);



//MPS Faults
//Fault if the beam is unsafe for current state
ffBeamParamsOK(i_xOK:=F_SafeBPCompare(i_stCurrentBeamParams, stLatchedBeamParams), 
				i_xReset:=i_xResetMPSFault,
				io_fbFFHWO := FastFaultOutput);

//Fault if the position is outside of the permitted range
ffActuatorBoundsOK(i_xOK := (lrPosition <= lrMPSUpperLimit AND lrPosition >= lrMPSLowerLimit), 
					i_xReset:=i_xResetMPSFault,
				io_fbFFHWO := FastFaultOutput);


	
//Collect all other faults
q_xFault := NOT ffBeamParamsOK.o_xFFLine OR
	NOT ffActuatorBoundsOK.o_xFFLine OR
	mcPower.Error	OR
	i_xMPSOverride	OR
	xInitFault;

//Any faults trip the fast fault line for this FB	
FastFaultOutput.CheckIn(NOT q_xFault);

END_FUNCTION_BLOCK

// ---- pmps-lib/MajorComponents/FB_FastFault.TcPOU
{attribute 'reflection'}
FUNCTION_BLOCK FB_FastFault
VAR_INPUT
	i_xOK		:	BOOL;
	i_xReset	:	BOOL; //resets when i_xOK is true and this is true
END_VAR
VAR_OUTPUT
	o_xFFLine	:	BOOL; //Connect to HW output or another FF input if you like
END_VAR
VAR_IN_OUT
	io_fbFFHWO		:	FB_HardwareFFOutput;
END_VAR
VAR
	{attribute 'instance-path'}
	{attribute 'noinit'}
	sPath	:	T_MaxString;
	
	xInit	:	BOOL :=TRUE;
	bsFF	:	RS;
	rtReset	:	R_TRIG;
	
END_VAR

IF xInit	THEN
	io_fbFFHWO.Register(i_sFFName:=sPath);
	//<TODO> if registration doesn't succeed, send warning to diagnostic
	xInit := FALSE;
END_IF


rtReset(CLK:=i_xReset);
bsFF(SET := rtReset.Q, RESET1:= NOT i_xOK);
o_xFFLine := bsFF.Q1;
io_fbFFHWO.CheckIn(bsFF.Q1);

END_FUNCTION_BLOCK

// ---- pmps-lib/HelperFunctions/F_DeviceState_To_DeviceStateExt.TcPOU
FUNCTION F_DeviceState_To_DeviceStateExt : ST_DeviceStateExt
VAR_INPUT
	stDeviceState	:	ST_DeviceState;
	xValid	:	BOOL;
END_VAR
VAR
END_VAR

F_DeviceState_To_DeviceStateExt.nStateRef := stDeviceState.nStateRef;
F_DeviceState_To_DeviceStateExt.rPosition	:=	stDeviceState.rPosition;
F_DeviceState_To_DeviceStateExt.rTolerance	:=	stDeviceState.rTolerance;
F_DeviceState_To_DeviceStateExt.sStateName	:= stDeviceState.sStateName;
F_DeviceState_To_DeviceStateExt.stReqBeamParam	:= stDeviceState.stReqBeamParam;
F_DeviceState_To_DeviceStateExt.xValid := xValid;

END_FUNCTION

// ---- pmps-lib/MajorComponents/BeamParameterTransitionManager.TcPOU
(*
Implements the procedure for safely transitioning between device states by asserting the correct beam parameters for 
the state *)
FUNCTION_BLOCK BeamParameterTransitionManager
VAR_IN_OUT
	
	fbArbiter	:	FB_Arbiter; //Connect to local arbiter
	
END_VAR
VAR_INPUT
	i_TransitionAssertionID	:	UDINT := 0;
	i_stTransitionAssertion : ST_BeamParams := PMPS_GVL_BeamParams.cstSafeBeam; //Assertion required during transition (always safer than anything inbetween)
	
	i_nRequestedAssertionID	:	UDINT := 0;
	i_stRequestedAssertion	:	ST_BeamParams := PMPS_GVL_BeamParams.cstSafeBeam; //Requested assertion, change whenever
	
	i_xMoving	:	BOOL := FALSE; //Provide rising edge when device begins moving <remove>
	i_xDoneMoving	:	BOOL := FALSE; //Provide rising edge when device is done with a move
	
	stCurrentBeamParameters	:	ST_BeamParams := PMPS_GVL_BeamParams.cstFullBeam; //Connect to current beam parameters
	
END_VAR
VAR_OUTPUT

	q_xTransitionAuthorized	:	BOOL := FALSE; //Rising edge indicating the device is safe to move, use as input to move execute (which requires a rising edge)

END_VAR

VAR
	nTargetAssertionID	:	UDINT := 0;
	stTargetAssertion	:	ST_BeamParams; //Current target assertion
	nCurrentAssertionID	:	UDINT := 0;
	
	xNewBP	:	BOOL;
	xTranBP	:	BOOL;
	xFinalBP	:	BOOL;
	
END_VAR

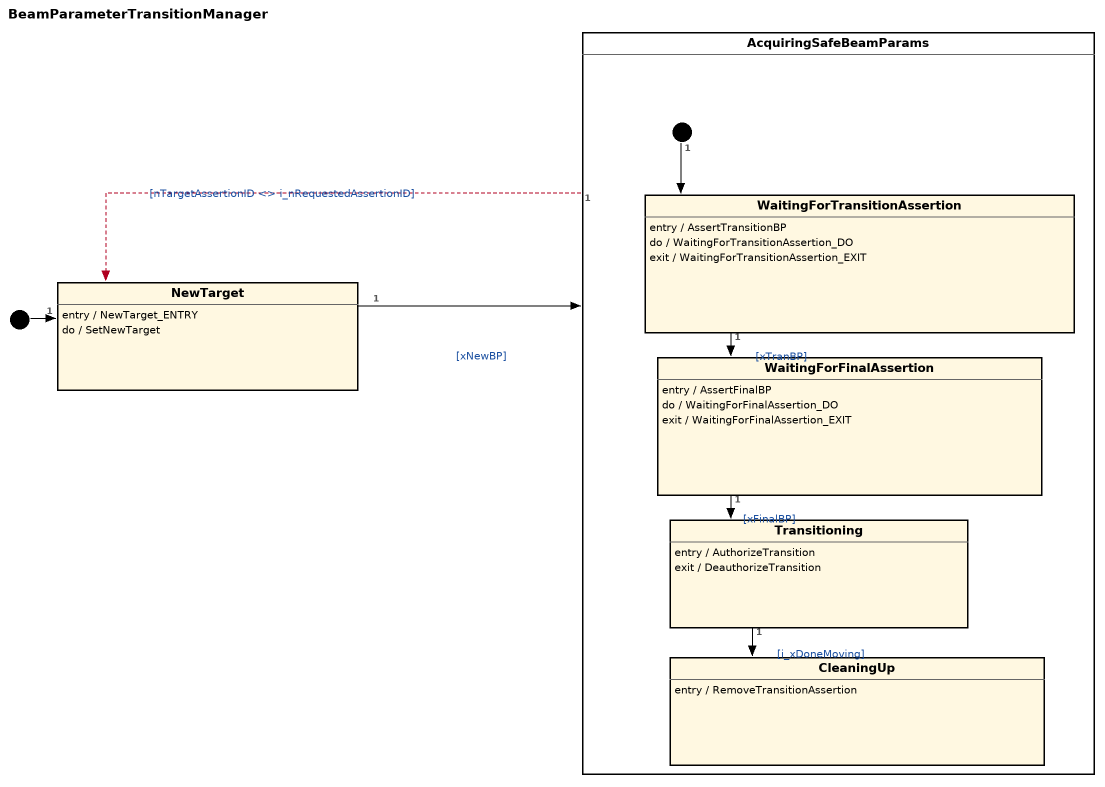
STATECHART BeamParameterTransitionManager  // abortable
    START StartState1_copy
    COMPOSITE STATE AcquiringSafeBeamParams
        START StartState1
        STATE WaitingForTransitionAssertion
            entry / AssertTransitionBP
            do / WaitingForTransitionAssertion_DO
            exit / WaitingForTransitionAssertion_EXIT
        STATE WaitingForFinalAssertion
            entry / AssertFinalBP
            do / WaitingForFinalAssertion_DO
            exit / WaitingForFinalAssertion_EXIT
        STATE Transitioning
            entry / AuthorizeTransition
            exit / DeauthorizeTransition
        STATE CleaningUp
            entry / RemoveTransitionAssertion
        StartState1 -> WaitingForTransitionAssertion  // priority 1, on completion
        WaitingForTransitionAssertion -> WaitingForFinalAssertion [xTranBP] // priority 1, rising edge
        WaitingForFinalAssertion -> Transitioning [xFinalBP] // priority 1, rising edge
        Transitioning -> CleaningUp [i_xDoneMoving] // priority 1, rising edge
    END_STATE
    STATE NewTarget
        entry / NewTarget_ENTRY
        do / SetNewTarget
    StartState1_copy -> NewTarget  // priority 1, on completion
    AcquiringSafeBeamParams -> NewTarget [nTargetAssertionID <> i_nRequestedAssertionID] // priority 1, exception
    NewTarget -> AcquiringSafeBeamParams [xNewBP] // priority 1
END_STATECHART

ACTION AcquiringSafeBeamParams_DO:
//xNewBP := nTargetAssertionID <> i_nRequestedAssertionID;
END_ACTION

ACTION AssertFinalBP:
//q_stFinalAssertion := stTargetAssertion;

//Clearing previous target parameters
(* This is considered safe at this step as the transition
state beam parameters should always be safer than the
current or target state beam parameters
*)
fbArbiter.RemoveRequest( nCurrentAssertionID );

//Asserting target parameters
fbArbiter.AddRequest(
	nTargetAssertionID,
	stTargetAssertion
);

//Remembering final assertionID for removal later
nCurrentAssertionID := nTargetAssertionID;
END_ACTION

ACTION AssertTransitionBP:

fbArbiter.AddRequest(
	i_TransitionAssertionID,
	i_stTransitionAssertion
);
END_ACTION

ACTION AuthorizeTransition:
q_xTransitionAuthorized := TRUE;
END_ACTION

ACTION DeauthorizeMove:

END_ACTION

ACTION DeauthorizeTransition:
q_xTransitionAuthorized := FALSE;
END_ACTION

ACTION NewTarget_ENTRY:
xNewBP := False;
END_ACTION

ACTION RemoveTransitionAssertion:
//q_stTransitionAssertion := PMPS_GVL_BeamParams.cstFullBeam;

//Removing transition assertion
fbArbiter.RemoveRequest( i_TransitionAssertionID );



//TODO add something to verify removal
END_ACTION

ACTION RemoveTransitionAuthorization:

END_ACTION

ACTION SetNewTarget:
IF i_nRequestedAssertionID <> 0 AND
	i_nRequestedAssertionID <> EXCLUDED_ASSERTION_ID THEN
	
	stTargetAssertion := i_stRequestedAssertion;
	nTargetAssertionID := i_nRequestedAssertionID;
	xNewBP := TRUE;
END_IF
END_ACTION

ACTION WaitingForFinalAssertion_DO:
//Final Assertion Verification

xFinalBP := F_SafeBPCompare(stCurrentBeamParameters, stTargetAssertion) AND
	fbArbiter.CheckRequest( i_nRequestedAssertionID);;
END_ACTION

ACTION WaitingForFinalAssertion_EXIT:
//Set this bool false so we can get a rising edge on the next try
xFinalBP := FALSE;
END_ACTION

ACTION WaitingForTransitionAssertion_DO:
//Transition Assertion Verification
xTranBP	:= F_SafeBPCompare(stCurrentBeamParameters, i_stTransitionAssertion) AND
	fbArbiter.CheckRequest(i_TransitionAssertionID);
END_ACTION

ACTION WaitingForTransitionAssertion_EXIT:
xTranBP := FALSE;
END_ACTION

END_FUNCTION_BLOCK

// ---- pmps-lib/HelperFunctions/F_SetStateParams.TcPOU
FUNCTION F_SetStateParams : BOOL;
VAR_INPUT
	nStateRef	:	UDINT;
	rPosition	:	REAL;
	rTolerance: REAL;
	stBeamParams	:	ST_BeamParams;
END_VAR
VAR_IN_OUT
	Table	:	FB_LinearDeviceStateTable;
END_VAR
VAR
	stDeviceState	:	ST_DeviceState;
	
END_VAR

stDeviceState.nStateRef := nStateRef;
stDeviceState.rPosition := rPosition;
stDeviceState.rTolerance := rTolerance;
stDeviceState.stReqBeamParam := stBeamParams;

Table.A_Add(
	key := nStateRef,
	putValue := stDeviceState
);

F_SetStateParams := Table.bOk;

END_FUNCTION

// ---- pmps-lib/MajorComponents/FB_LinearDeviceStateTable.TcPOU
(* This function block implements simple database. Data element values are stored in the hash table.  *)
FUNCTION_BLOCK FB_LinearDeviceStateTable
VAR_INPUT
	key 		: DWORD := 0;(* Entry key: used by A_Lookup, A_Remove method, the key variable is also used by A_Add method *)
	putPosPtr	: POINTER TO T_HashTableEntry := 0;(* Hash table entry position pointer (used by A_Find, A_GetNext, A_GetPrev) *)
	putValue 	: ST_DeviceState;(* Hash table entry value (used by A_AddHead, A_AddTail, A_Find )*)
END_VAR
VAR_OUTPUT
	bOk			: BOOL := FALSE;(* TRUE = Success, FALSE = Failed *)
	getPosPtr	: POINTER TO T_HashTableEntry := 0;(* Returned hash table entry position pointer *)
	getValue 	: ST_DeviceState;(* Returned hash table entry value *)
	nCount		: UDINT := 0;(* Hash table size (number of used entries, used by A_Count) *)
END_VAR
VAR
	dataPool	: ARRAY[0..MAX_DEVICE_STATES] OF ST_DeviceState;(* Structured data element pool *)
	entries		: ARRAY[0..MAX_DEVICE_STATES] OF T_HashTableEntry;(* Max. number of hash table entries. The value of table entry = 32 bit integer (pointer to dataPool-array-entry) *)
	fbTable 	: FB_HashTableCtrl;(* basic hash table control function block *)
	hTable 		: T_HHASHTABLE;(* hash table handle *)
	pRefPtr		: POINTER TO ST_DeviceState := 0;
	indexOfElem	: ULINT;(* Integer value (max. size: x86=>32bit, x64=>64bit)*)
END_VAR

;

ACTION A_Add:
(* Adds entry to the table *)
MEMSET( ADR( getValue ), 0, SIZEOF( getValue ) );
getPosPtr := 0;

fbTable.A_Add( hTable := hTable, key := key, putValue := ADR(PMPS_GVL_BeamParams.cstSafeBeam)(* we will set this value later *), getPosPtr=>getPosPtr, bOk=>bOk );(* Add new element to the table, getPosPtr points to the new entry *)
IF fbTable.bOk THEN(* Success *)
	fbTable.A_GetIndexAtPosPtr( hTable := hTable, putPosPtr := getPosPtr, getValue =>indexOfElem, bOk=>bOk );(* Get array index of getPosPtr entry *)
	IF fbTable.bOk THEN(* Success *)
		pRefPtr 	:= ADR( dataPool[indexOfElem] );(* Get pointer to the data element *)

		pRefPtr^ := putValue;(* copy application value *)

		fbTable.A_Add( hTable := hTable, key := key, putValue := pRefPtr, bOk=>bOk );(* Assign the entry value = pointer to the data element *)
		IF fbTable.bOk THEN(* Success *)
			getValue := putValue;
		END_IF
	END_IF
END_IF
END_ACTION

ACTION A_Count:
(* Count number of used entries *)
nCount := hTable.nCount;
bOk := TRUE;
END_ACTION

ACTION A_GetFirst:
(* Get first entry position pointer and value *)
MEMSET( ADR( getValue ), 0, SIZEOF( getValue ) );
getPosPtr := 0;

fbTable.A_GetFirst( hTable := hTable, putPosPtr := putPosPtr, getValue=>pRefPtr, getPosPtr=>getPosPtr, bOk=>bOk );
IF fbTable.bOk THEN
	getValue := pRefPtr^;
END_IF
END_ACTION

ACTION A_GetNext:
(* Get next entry position pointer and value *)
MEMSET( ADR( getValue ), 0, SIZEOF( getValue ) );
getPosPtr := 0;
bOk := FALSE;

IF putPosPtr = 0 THEN
	RETURN;
END_IF

fbTable.A_GetNext( hTable := hTable, putPosPtr := putPosPtr, getValue=>pRefPtr, getPosPtr=>getPosPtr, bOk=>bOk );
IF fbTable.bOk THEN
	getValue := pRefPtr^;
END_IF
END_ACTION

ACTION A_Lookup:
(* Lookup for entry by key  *)
MEMSET( ADR( getValue ), 0, SIZEOF( getValue ) );
getPosPtr := 0;

fbTable.A_Lookup( key := key, hTable := hTable, putPosPtr := putPosPtr, getValue=>pRefPtr, getPosPtr=>getPosPtr, bOk=>bOk );
IF fbTable.bOk THEN
	getValue := pRefPtr^;
END_IF
END_ACTION

ACTION A_Remove:
(* Search for entry and remove it *)
MEMSET( ADR( getValue ), 0, SIZEOF( getValue ) );
getPosPtr := 0;

fbTable.A_Remove( key := key, hTable := hTable, putPosPtr := putPosPtr, getValue=>pRefPtr, getPosPtr=>getPosPtr, bOk=>bOk );
IF fbTable.bOk THEN
	getValue := pRefPtr^;
END_IF
END_ACTION

ACTION A_Reset:
(* Reset/initialize linked list *)
MEMSET( ADR( getValue ), 0, SIZEOF( getValue ) );
getPosPtr := 0;
bOk := F_CreateHashTableHnd( ADR( entries ), SIZEOF( entries ), hTable );(* Intialize table handle *)
fbTable.A_Reset( hTable := hTable, bOk=>bOk );
nCount := 0;
END_ACTION

END_FUNCTION_BLOCK

// ---- POUs/Fast_Faults_Setup.TcPOU
// Run at the start of each cycle

PROGRAM Fast_Faults_Setup
VAR
END_VAR

g_FastFaultOutput1();

END_PROGRAM

// ---- POUs/PMPS_Arbiter.TcPOU
PROGRAM PMPS_Arbiter
VAR
	
	
	
	
	fbPhotonEnergyWatcher	:	FB_PhotonEnergyWatcher;
	
	//fbMPSInterface	:	FB_BeamClassOutputs;
	
	{attribute 'TcLinkTo' := '.i_stBP:=TIIB[PMPS_IF]^IO Inputs^CurrentBP1;.xTxPDO_toggle:=TIIB[PMPS_IF]^SYNC Inputs^TxPDO toggle;.xTxPDO_state:=TIIB[PMPS_IF]^SYNC Inputs^TxPDO state'}
	fbBPFanout	:	FB_BeamParamFanout;
	
	{attribute 'TcLinkTo' := '.i_stBP:=TIIB[PMPS_IF]^IO Outputs^ReqBP'}
	q_stReqBeamParams	AT %Q*	:	ST_BeamParams;
	
	//fbBPFanout1	:	FB_BeamParamFanout_1;
	
	fbBPRequestor	:	FB_BPRequestor;
	fbSimAttenuator :	FB_AttenuatorSimulator;
	
	stCurrentBeamParam	AT %I*	:	ST_BeamParams;
	
END_VAR

PMPS_GVL_BeamParams.stCurrentBeamParameters.neVRange := F_eVRangeCalculator(
	PMPS_GVL_BeamParams.stCurrentBeamParameters.reV,
	PMPS_GVL_BeamParams.stCurrentBeamParameters.neVRange);

//Example with attenuator peel-off
//////////////////////////////////

//Beam parameter requestor
fbBPRequestor(stReqBP := g_fbArbiter1.GetArbitratedBP(),
q_ReqAtt=>fbSimAttenuator.i_rRequestedAttenuation,
q_stReqBP=>q_stReqBeamParams);

//Request beam class
//fbMPSInterface();

//Keep an eye on the photon energy
fbPhotonEnergyWatcher(i_stCurrentBeamParams	:= PMPS_GVL_BeamParams.stCurrentBeamParameters,
					i_stRequestedBeamParams := fbBPRequestor.q_stReqBP,
					io_fbFFHWO:= GVL.g_FastFaultOutput1);



fbSimAttenuator(Arbiter:=g_fbArbiter2);


//Beam parameter fanout
//fbBPFanout();

END_PROGRAM

// ---- pmps-lib/MajorComponents/FB_PhotonEnergyWatcher.TcPOU
(*
A. Wallace 2019-4-22
The photon energy watcher ensures the current and target photon energy is within
the arbirated bounds. Target in this case means, the calculated target photon energy
from the PVs that control the mechatronics of the undulators/ the electron energy.

If there are control PVs that match the monitor PVs, the control PVs are used to 
calculate a "target" photon energy. This is supposed to cover when the undulators/
electron energy is transitioning.

The abritrated bounds come from a simple AND of all the permitted ranges. See
the arbitrate action of the arbiter FB.

Note, this protection logic does not account for beam-off when determining fast-fault
status. If a device is requesting a limited range of eV, this request must be honored,
regardless of current beam-rate.
*)
FUNCTION_BLOCK FB_PhotonEnergyWatcher
VAR_INPUT
	i_stCurrentBeamParams	:	ST_BeamParams; //Link to global beam params
	i_stMachineTargetBeamParams	:	ST_BeamParams; //Link to global machine target beam params
	i_stRequestedBeamParams	:	ST_BeamParams; //Link to arbiter output or beam param. requestor
	// Reset fault
	i_xReset: BOOL;
END_VAR
VAR_OUTPUT
END_VAR
VAR_IN_OUT
	io_fbFFHWO	:	FB_HardwareFFOutput;
END_VAR
VAR
	xPhotonEnergyWithinBounds	:	BOOL;
	fbFF	:	FB_FastFault;
END_VAR

xPhotonEnergyWithinBounds := (i_stCurrentBeamParams.neVRange AND i_stRequestedBeamParams.neVRange) = i_stCurrentBeamParams.neVRange;

fbFF(i_xOK := xPhotonEnergyWithinBounds,
	i_xReset := i_xReset,
	io_fbFFHWO := io_fbFFHWO);

END_FUNCTION_BLOCK

// ---- pmps-lib/MajorComponents/FB_BeamParamFanout.TcPOU
FUNCTION_BLOCK FB_BeamParamFanout
VAR_INPUT

END_VAR
VAR_OUTPUT
	stBP	:	ST_BeamParams;
END_VAR
VAR
	i_stBP	AT %I* :	ST_BeamParams;
	
	xTxPDO_toggle	AT 	%I* :	BIT;
	xTxPDO_state	AT	%I*	:	BIT;
END_VAR



stBP.xValidToggle;

END_FUNCTION_BLOCK

// ---- pmps-lib/MajorComponents/FB_BPRequestor.TcPOU
FUNCTION_BLOCK FB_BPRequestor
VAR_INPUT
	stReqBP	:	ST_BeamParams;
END_VAR
VAR_OUTPUT
	q_stReqBP :	ST_BeamParams;
	q_ReqAtt  : REAL;
END_VAR
VAR
	
END_VAR

q_stReqBP := stReqBP;
q_ReqAtt := stReqBP.fAtt;

END_FUNCTION_BLOCK

// ---- pmps-lib/TestComponents/FB_AttenuatorSimulator.TcPOU
FUNCTION_BLOCK FB_AttenuatorSimulator
VAR_INPUT
	i_rRequestedAttenuation	:	REAL;
	i_stBPReadback	:	ST_BeamParams;
END_VAR
VAR_OUTPUT
	q_xFault	:	BOOL;
	q_rCurrentAttenuation	:	REAL;
END_VAR
VAR_IN_OUT
	Arbiter	:	FB_Arbiter; //Higher level arbiter from which upstream attenuation can be requested
END_VAR
VAR
	tonDelay	:	TON := (
		PT := T#3S
		);
END_VAR

// Really basic delay
tonDelay(IN := i_rRequestedAttenuation <> q_rCurrentAttenuation);

IF tonDelay.Q THEN
	q_rCurrentAttenuation := i_rRequestedAttenuation;
END_IF

END_FUNCTION_BLOCK

// ---- pmps-lib/HelperFunctions/F_eVRangeCalculator.TcPOU
(*
A. Wallace 2019-8-8

Provides bit range of eV.
*)
FUNCTION F_eVRangeCalculator : WORD // Bit-range of current photon energy
VAR_INPUT
	reV	:	REAL; // Photon energy
	LastWord	:	WORD; // Range word of previous cycle
END_VAR
VAR
	nIndex: INT;
	RangeWord: WORD;
	rPreviousBoundary: REAL := 0;
	rHyst: REAL := 0.05; // <TODO> global constant
	MaxEv	:	REAL := PMPS_GVL_BeamParams.g_areVBoundaries[PMPS_GVL_BeamParams.g_cBoundaries]*1000;
END_VAR


IF reV < 0 THEN F_eVRangeCalculator := 16#FFFF; RETURN; END_IF

FOR nIndex := 0 TO PMPS_GVL_BeamParams.g_cBoundaries DO
	
	// If previously active then check if it should be cleared
	IF LastWord.0 THEN 
		// Hysteresis condition
		IF (reV > MIN(PMPS_GVL_BeamParams.g_areVBoundaries[nIndex]*1000 + rHyst*1000, MaxEv) ) OR
		(reV < MAX(rPreviousBoundary*1000 - rHyst*1000, 0) ) THEN
			RangeWord.0 := 0; // If out of range of hys. mark inactive
		ELSE
			RangeWord.0 := 1;
		END_IF
	ELSE // Check if we should mark as active
		IF (reV <= PMPS_GVL_BeamParams.g_areVBoundaries[nIndex]*1000) AND
		(reV >= rPreviousBoundary*1000) THEN
			RangeWord.0 := 1;
		END_IF
	END_IF
	
	// Catch if the hysteresis is set too large for the range
	IF rPreviousBoundary + rHyst >= PMPS_GVL_BeamParams.g_areVBoundaries[nIndex] THEN
		RangeWord.0 := 1; // Setting the bit true here as a failsafe
		//<TODO> Add major error or warning here
	END_IF
	
	rPreviousBoundary := PMPS_GVL_BeamParams.g_areVBoundaries[nIndex];
	// Shift to next bit
	RangeWord := ROR(RangeWord, 1);
	LastWord := SHR(LastWord, 1);
	
END_FOR

F_eVRangeCalculator := RangeWord;

END_FUNCTION

// ---- POUs/Fast_Faults_Evaluate.TcPOU
PROGRAM Fast_Faults_Evaluate
VAR
END_VAR

g_FastFaultOutput1.EvaluateOutput();

END_PROGRAM

// ---- POUs/MachineSimulation.TcPOU
PROGRAM MachineSimulation
VAR
	fbMachine	:	FB_MachineSimulator;
	
	i_SimReqBP	AT	%I*	:	ST_BeamParams;
	q_SimCurrBP	AT %Q*	:	ST_BeamParams;
END_VAR

//Machine simulator
fbMachine(
	i_stAssertedParams := i_SimReqBP,
	q_stMachineParams => PMPS_GVL_BeamParams.stCurrentBeamParameters,
	i_xFault	:= NOT GVL.g_FastFaultOutput1.q_xFastFaultOut
	);
	
q_SimCurrBP	:= fbMachine.q_stMachineParams;
q_SimCurrBP.neVRange := i_SimReqBP.neVRange;

END_PROGRAM

// ---- pmps-lib/TestComponents/FB_MachineSimulator.TcPOU
(* Simulates the machine responding to requests by adding a bit of delay/ ramps
*)
FUNCTION_BLOCK FB_MachineSimulator
VAR_INPUT
	i_stAssertedParams	:	ST_BeamParams;
	i_reV	:	REAL;
	i_xFault	:	BOOL;
END_VAR
VAR_OUTPUT
	q_stMachineParams	:	ST_BeamParams;
END_VAR
VAR
	fTargetAtt: REAL;
	tonAttTimer	:	TON := (
		PT := T#2S
		);
	fTargetPP_mJ: REAL;
	tonPPETimer: TON := (
		PT := T#2S
	);
END_VAR


//Attenuation
IF i_stAssertedParams.fAtt <> fTargetAtt THEN
	tonAttTimer(IN:=FALSE);
	fTargetAtt := i_stAssertedParams.fAtt;
ELSIF NOT tonAttTimer.Q THEN
	tonAttTimer(IN:=TRUE);
ELSE
	q_stMachineParams.fAtt := fTargetAtt;
END_IF

//Pulse Energy
IF i_stAssertedParams.fPP_mJ <> fTargetPP_mJ THEN
	tonPPETimer(IN:=FALSE);
	fTargetPP_mJ := i_stAssertedParams.fPP_mJ;
ELSIF NOT tonAttTimer.Q THEN
	tonPPETimer(IN:=TRUE);
ELSE
	q_stMachineParams.fPP_mJ := fTargetPP_mJ;
END_IF

//Photon Energy is set arbitrarily, beyond our control.
q_stMachineParams.reV := i_reV;

//Rate
IF i_xFault THEN
	q_stMachineParams.nRate := 0;
ELSE
	q_stMachineParams.nRate := i_stAssertedParams.nRate;
END_IF

END_FUNCTION_BLOCK

// ---- POUs/TestSetups.TcPOU
//Test setups (fixtures), for PMPS components
PROGRAM TestSetups
VAR
	fbBPTMTest	:	FB_BPTM_Test;
	fbSafeBPCompareTest	:	FB_SafeBPCompare_Test;
	fbevWithinSpecTest	:	FB_evWithinSpec_Test;
	fbPEWTest	:	FB_PhotonEnergyWatcher_Test;
	fbFFTest	:	FB_FastFault_Test;
	fbArbiterTest	:	FB_Arbiter_Test;
END_VAR

TcUnit.RUN();

END_PROGRAM

// ---- pmps-lib/TestComponents/FB_BPTM_Test.TcPOU
{attribute 'call_after_init'}
FUNCTION_BLOCK FB_BPTM_Test EXTENDS TcUnit.FB_TestSuite
VAR_INPUT
END_VAR
VAR_OUTPUT
END_VAR
VAR
END_VAR

BPTMBasicFunction();

METHOD BPTMBasicFunction
VAR_INPUT
END_VAR
VAR	
	//Final and transition assertions
	nTransitionID	:	UDINT := 1;
	stTransitionAssertion	:	ST_BeamParams := PMPS_GVL_BeamParams.cstSafeBeam;
	
 	nReqID	:	UDINT	:= 2;
	stReqAssertion	:	ST_BeamParams := PMPS_GVL_BeamParams.cstSafeBeam;
	
	fbMachine	:	FB_MachineSimulator;	
	
END_VAR
VAR_INST
	fbBPTM_TestBasicFunction	:	BeamParameterTransitionManager;
	fbArbiter	:	FB_Arbiter;
	xFirstPass	:	BOOL := TRUE;
	eTestStep: eBPTMTestStates := eBPTMTestStates.Init;
END_VAR
CASE eTestStep OF

eBPTMTestStates.Init:
	fbArbiter.A_Init();
	
	eTestStep := eBPTMTestStates.WaitingForTransitionAssertion;

eBPTMTestStates.WaitingForTransitionAssertion:
	TEST('BPTMBasicFunction');
	
	//Call BPTM with requested final state and transition state
	fbBPTM_TestBasicFunction(
		fbArbiter := fbArbiter,
		i_TransitionAssertionID := nTransitionID,
		i_stTransitionAssertion := stTransitionAssertion,
		
		i_nRequestedAssertionID := nReqID,
		i_stRequestedAssertion := stReqAssertion
	);
	
	IF fbBPTM_TestBasicFunction.UML_SC_BeamParameterTransitionManager.States
	[fbBPTM_TestBasicFunction.UML_SC_BeamParameterTransitionManager.Names.WaitingForTransitionAssertion].Active THEN
	
		AssertTrue(fbArbiter.CheckRequest(nTransitionID), 'Arbiter did not accept BPTM transition assertion');
		
		AssertFalse(fbArbiter.CheckRequest(nReqID), 'Arbiter has requested too early.');
				
		AssertFalse(fbBPTM_TestBasicFunction.q_xTransitionAuthorized,
			'Transition should not be authorized until the arbiter has final assertion');
			
		TEST_FINISHED_NAMED('BPTMBasicFunction');
		
		eTestStep := eBPTMTestStates.WaitingForFinalAssertion;
	END_IF

eBPTMTestStates.WaitingForFinalAssertion:

	TEST('BPTM Requests Final');
	fbBPTM_TestBasicFunction(fbArbiter := fbArbiter,
		stCurrentBeamParameters := stTransitionAssertion);
	
	IF fbBPTM_TestBasicFunction.UML_SC_BeamParameterTransitionManager.States
	[fbBPTM_TestBasicFunction.UML_SC_BeamParameterTransitionManager.Names.WaitingForFinalAssertion].Active THEN
	
		AssertTrue(fbArbiter.CheckRequest(nReqID),
			'Transition assertion should be in arbiter');
		
		AssertTrue(fbArbiter.CheckRequest(nReqID),
			'Final assertion should be in arbiter');
			
		AssertFalse(fbBPTM_TestBasicFunction.q_xTransitionAuthorized,
			'Transition should not be authorized until the arbiter has final assertion');
			
		TEST_FINISHED_NAMED('BPTM Requests Final');
	
		eTestStep := eBPTMTestStates.Transitioning;
	END_IF

eBPTMTestStates.Transitioning:
	TEST('BPTM Authorizes Transition');
	fbBPTM_TestBasicFunction(fbArbiter := fbArbiter,
		stCurrentBeamParameters := stTransitionAssertion);
		
	IF fbBPTM_TestBasicFunction.UML_SC_BeamParameterTransitionManager.States
	[fbBPTM_TestBasicFunction.UML_SC_BeamParameterTransitionManager.Names.Transitioning].Active THEN
	
		AssertTrue(fbArbiter.CheckRequest(nReqID),
			'Transition assertion should be in arbiter');
		
		AssertTrue(fbArbiter.CheckRequest(nReqID),
			'Final assertion should be in arbiter');
			
		AssertTrue(fbBPTM_TestBasicFunction.q_xTransitionAuthorized,
			'Transition should be authorized at this point.');
			
		AssertEquals(nReqID, fbBPTM_TestBasicFunction.nCurrentAssertionID,
			'nCurrentAssertionID not set.');
	
		TEST_FINISHED_NAMED('BPTM Authorizes Transition');
	END_IF

eBPTMTestStates.CleaningUp:	
	
END_CASE
(*	
TEST('BPTM Authorizes Transition');
AssertTrue(fbBPTM.q_xTransitionAuthorized,
	'Transition should be authorized at this point');
TEST_FINISHED();
	
TEST('BPTM Current assertion id is set');
AssertEquals(nReqID, fbBPTM.nCurrentAssertionID,
	'nCurrentAssertionID not set.');
TEST_FINISHED();
	
TEST('BPTM Transition Deauthorized');
fbBPTM(fbArbiter := fbArbiter,
		i_xDoneMoving := TRUE);
AssertFalse(fbBPTM.q_xTransitionAuthorized,
	'Transition authorization should go away when done moving');
TEST_FINISHED();
	
TEST('BPTM Transition BP request removed');
AssertFalse(fbArbiter.CheckRequest(nTransitionID),
	'Transition ID still in arbiter');
	
//Basic testing is complete, interruption functionality testing next
//Continuing to use the same BPTM because internal variable nCurrentAssertionID is now non-zero

TEST_FINISHED();*)
END_METHOD

END_FUNCTION_BLOCK

// ---- pmps-lib/TestComponents/FB_SafeBPCompare_Test.TcPOU
{attribute 'call_after_init'}
FUNCTION_BLOCK FB_SafeBPCompare_Test EXTENDS TcUnit.FB_TestSuite
VAR_INPUT
END_VAR
VAR_OUTPUT
END_VAR
VAR

END_VAR

BeamOffIsSafe();
BPComparisonCheck();

//Verify beam off is considered safe.
METHOD BeamOffIsSafe
VAR_INPUT
END_VAR
VAR
	stBeamOn	:	ST_BeamParams;
	stBeamOff	:	ST_BeamParams;
	
END_VAR
stBeamOn := F_SetBeamParams(
	50, //50% attenuation is more conservative than 0
	10,
	16#FFFF,
	120);

stBeamOff := F_SetBeamParams(
	0, //0% attenuation
	10,
	16#FFFF,
	0); //0 beam rate means this bps is actually safer than BeamOn

TEST('BeamOffIsSafe');
	
AssertTrue(
	F_SafeBPCompare(stBeamOff, stBeamOn),
	'SafeBPCompare does not think beam rate = 0 is safer than anything else.'); 
TEST_FINISHED();
END_METHOD

//Verify BP comparison remains logical.
METHOD BPComparisonCheck
VAR_INPUT
END_VAR
VAR
	stSafer	:	ST_BeamParams;
	stNotSoSafe	:	ST_BeamParams;
END_VAR
TEST('BPComparisonCheck');


//Attenuation
stSafer := F_SetBeamParams(
	1, //
	10,
	16#FFFF,
	1);

stNotSoSafe := F_SetBeamParams(
	0, //
	10,
	16#FFFF,
	1); 
	
AssertTrue(
	F_SafeBPCompare(stSafer, stNotSoSafe),
	'Attenuation eval is broken (True)'); 

AssertFalse(
	F_SafeBPCompare(stNotSoSafe, stSafer),
	'Attenuation eval is broken (False)');
	
	
//Rate
stSafer := F_SetBeamParams(
	0,
	10,
	16#FFFF,
	1); //

stNotSoSafe := F_SetBeamParams(
	0,
	10,
	16#FFFF,
	10); //
	
AssertTrue(
	F_SafeBPCompare(stSafer, stNotSoSafe),
	'Rate eval is broken (True)'); 

AssertFalse(
	F_SafeBPCompare(stNotSoSafe, stSafer),
	'Rate eval is broken (False)');
	
//Pulse energy
stSafer := F_SetBeamParams(
	0, 
	1, //
	16#FFFF,
	1);

stNotSoSafe := F_SetBeamParams(
	0, 
	10, //
	16#FFFF,
	1); 
	
AssertTrue(
	F_SafeBPCompare(stSafer, stNotSoSafe),
	'Pulse energy eval is broken (True)'); 

AssertFalse(
	F_SafeBPCompare(stNotSoSafe, stSafer),
	'Pulse energy eval is broken (False)');	
	
//Photon energy
//More extensive tests elsewhere
stSafer := F_SetBeamParams(
	0, 
	1, 
	2#0000_0000_0000_0110, //200-400eV
	1);
	
stSafer.reV := 300; //

stNotSoSafe := F_SetBeamParams(
	0, 
	1, 
	2#0000_0000_0000_0110, //200-400ev
	1);
	
stNotSoSafe.reV := 401;
	
AssertTrue(
	F_SafeBPCompare(stSafer, stNotSoSafe),
	'Photon energy eval is broken (True)'); 

AssertFalse(
	F_SafeBPCompare(stNotSoSafe, stSafer),
	'Photon energy eval is broken (False)');	
TEST_FINISHED();
END_METHOD

END_FUNCTION_BLOCK

// ---- pmps-lib/TestComponents/FB_eVWithinSpec_Test.TcPOU
{attribute 'call_after_init'}
FUNCTION_BLOCK FB_eVWithinSpec_Test EXTENDS TcUnit.FB_TestSuite
VAR_INPUT
END_VAR
VAR_OUTPUT
END_VAR
VAR
END_VAR

evWithinRangeChecks();

METHOD evWithinRangeChecks
VAR_INPUT
END_VAR
VAR

END_VAR
TEST('evWithinRangeChecks');
	
//Upper limit equal
AssertTrue(
	F_eVWithinSpec(300, 2#0000_0000_0000_0010),
	'Upper limit not inclusive');
//Lower limit equal
AssertTrue(
	F_eVWithinSpec(300, 2#0000_0000_0000_0100),
	'Lower limit not inclusive');
//Out of range
AssertFalse(
	F_eVWithinSpec(300.1, 2#0000_0000_0000_0010),
	'Out of range failed, whatever you did, it broke this really bad.');
//Negative eV
AssertFalse(
	F_eVWithinSpec(-300, 16#FFFF),
	'Working with antimatter? Negative eV should not be acceptable.');
//Upper unallocated range
AssertFalse(
	F_eVWithinSpec(1701, 2#1000_0000_0000_0000),
	'eV range should not evaluate past 1.7keV');
	
TEST_FINISHED();
END_METHOD

END_FUNCTION_BLOCK

// ---- pmps-lib/HelperFunctions/F_eVWithinSpec.TcPOU
//reV must be within permitted range.
FUNCTION F_eVWithinSpec : BOOL
VAR_INPUT
	reV	:	REAL;	//Photon energy to check if within permitted range
	nPermittedRange	:	WORD; //Permitted range
END_VAR
VAR
	//Holding register for permitted ranges
	nPermittedRangeHolding	:	WORD; 
	//For loop counter
	nIndex	:	INT;
	// Lower boundary for range check 
	rPreviousBoundary: REAL := 0;
END_VAR

(* How this works:
The within range bool is initialized to false.
Load the word representation of ranges into a holding register.
If the bit at position zero of the holding register is true, and the input eV is
below the boundary at the index position of the boundary array, and the previous boundary
(which initializes at 0), then the within range bool is set. 
Then, we stash the upper boundary as the lower boundary for the next comparison,
and shift the holding register right, which moves the next bit to the zero position.
*)
nPermittedRangeHolding := nPermittedRange;

FOR nIndex := 0 TO PMPS_GVL_BeamParams.g_cBoundaries DO
		
	F_eVWithinSpec S= nPermittedRangeHolding.0 AND( 
		(reV <= PMPS_GVL_BeamParams.g_areVBoundaries[nIndex]*1000) AND
		(reV >= rPreviousBoundary*1000) );
		
	IF F_eVWithinSpec THEN RETURN; END_IF
	
	rPreviousBoundary := PMPS_GVL_BeamParams.g_areVBoundaries[nIndex];
	nPermittedRangeHolding := SHR(nPermittedRangeHolding, 1);
END_FOR

END_FUNCTION

// ---- pmps-lib/TestComponents/FB_PhotonEnergyWatcher_Test.TcPOU
{attribute 'call_after_init'}
FUNCTION_BLOCK FB_PhotonEnergyWatcher_Test EXTENDS TcUnit.FB_TestSuite
VAR_INPUT
END_VAR
VAR_OUTPUT
END_VAR
VAR

END_VAR

PEWatcherBasicFunction();

METHOD PEWatcherBasicFunction
VAR_INPUT
END_VAR
VAR
	fbPEW	:	FB_PhotonEnergyWatcher;
	fbFFO	:	FB_HardwareFFOutput;
	q_Output	:	BOOL;
	
	stCurBeamParams	:	ST_BeamParams;
	stMachineTargetBeamParams	:	ST_BeamParams;
	stReqBeamParams	:	ST_BeamParams;
END_VAR
TEST('PEWatcherBasicFunction');

//Clear FFO fault to start
fbFFO(i_xReset:=TRUE);

//All eV OK
stCurBeamParams.reV := 800;
	
stMachineTargetBeamParams.reV := 800;

stReqBeamParams.neVRange := 2#1111_1111_1111_1111;	

fbFFO(i_xReset:=FALSE); //Reset request released
	
fbPEW(i_stCurrentBeamParams := stCurBeamParams,
	i_stMachineTargetBeamParams := stMachineTargetBeamParams,
	i_stRequestedBeamParams := stReqBeamParams,
	io_fbFFHWO := fbFFO,
	i_xReset := TRUE); //Clear local FF within PEW
	
fbFFO.EvaluateOutput(q_xFastFaultOut=>q_Output); //This simulates a completed PLC cycle
//Evaluate output should be called once at the end of a PLC cycle.

AssertTrue(q_Output,
	'Beam within limits, FFO should be true');
	
	
//Req eV moved out of range
stCurBeamParams.reV := 800;
	
stMachineTargetBeamParams.reV := 800;

stReqBeamParams.neVRange := 2#0000_1111_0011_1111;

fbPEW.i_xReset := FALSE; //release local FF reset req	
fbPEW(i_stCurrentBeamParams := stCurBeamParams,
	i_stMachineTargetBeamParams := stMachineTargetBeamParams,
	i_stRequestedBeamParams := stReqBeamParams,
	io_fbFFHWO := fbFFO);
	
fbFFO.EvaluateOutput(q_xFastFaultOut=>q_Output);

AssertFalse(q_Output,
	'Limits moved beyond current and target beam, should produce a fault.');

//Beam and target eV moved back within permitted ranges, reset clears fault
stCurBeamParams.reV := 300;
	
stMachineTargetBeamParams.reV := 300;

stReqBeamParams.neVRange := 2#0000_1111_0011_1111;

fbFFO(i_xReset:=TRUE); //New reset request

fbPEW.i_xReset := TRUE; //New reset request

fbPEW(i_stCurrentBeamParams := stCurBeamParams, //Beam params are now within spec
	i_stMachineTargetBeamParams := stMachineTargetBeamParams,
	i_stRequestedBeamParams := stReqBeamParams,
	io_fbFFHWO := fbFFO);
	
fbFFO.EvaluateOutput(q_xFastFaultOut=>q_Output);

AssertTrue(q_Output,
	'Beam within limits after reset, FFO should be true');
	
//At this point, the fast fault would be cleared

//Current beam eV moved out of range
stCurBeamParams.reV := 800; //Moved out of range
	
stMachineTargetBeamParams.reV := 300; //Still within range

stReqBeamParams.neVRange := 2#0000_1111_0011_1111;

fbPEW(i_stCurrentBeamParams := stCurBeamParams,
	i_stMachineTargetBeamParams := stMachineTargetBeamParams,
	i_stRequestedBeamParams := stReqBeamParams,
	io_fbFFHWO := fbFFO);
	
fbFFO.EvaluateOutput(q_xFastFaultOut=>q_Output);

AssertFalse(q_Output,
	'Current beam moved beyond set limits, should produce a fault');

//Target beam eV moved out of range
fbFFO(i_xReset:=FALSE); //Reset released
fbFFO(i_xReset:=TRUE); //New reset request comes in at the top of a cycle, but will be overridden

stCurBeamParams.reV := 300; //Now within range
	
stMachineTargetBeamParams.reV := 800; //Moved out of range

stReqBeamParams.neVRange := 2#0000_1111_0011_1111;

fbPEW.i_xReset := TRUE; //Attempt to reset local FF will fail
fbPEW(i_stCurrentBeamParams := stCurBeamParams,
	i_stMachineTargetBeamParams := stMachineTargetBeamParams,
	i_stRequestedBeamParams := stReqBeamParams,
	io_fbFFHWO := fbFFO);
	
fbFFO.EvaluateOutput(q_xFastFaultOut=>q_Output);

AssertFalse(q_Output,
	'Target beam moved beyond set limits, should produce a fault');
	
TEST_FINISHED();
END_METHOD

END_FUNCTION_BLOCK

// ---- pmps-lib/TestComponents/FB_FastFault_Test.TcPOU
{attribute 'call_after_init'}
FUNCTION_BLOCK FB_FastFault_Test EXTENDS TcUnit.FB_TestSuite
VAR_INPUT
END_VAR
VAR_OUTPUT
END_VAR
VAR

END_VAR

FFCombinedFunctionality();
FFRegistration();

METHOD FFCombinedFunctionality
VAR_INPUT
END_VAR
VAR
	fbFF	:	FB_FastFault;
	fbFFO	:	FB_HardwareFFOutput;
	
END_VAR
TEST('FFCombinedFunctionality');

//Clear initial faults
fbFFO(i_xReset:=TRUE); //Reset requested at start of cycle

fbFF(io_fbFFHWO := fbFFO, //FF reset somehwere in code
	i_xOK := TRUE,
	i_xReset := TRUE);

fbFFO.EvaluateOutput(); //FFO eval called at end of cycle
	
AssertTrue(fbFFO.q_xFastFaultOut,
	'Fast fault did not clear');


//Induce fault with FF

fbFFO(i_xReset := FALSE); //Reset released at start of cycle

fbFF(io_fbFFHWO := fbFFO, //FF faulted
	i_xOK := FALSE); //Reset is still set true from last call.
	
fbFFO.EvaluateOutput(); //FFO eval called at end of cycle

AssertFalse(fbFFO.q_xFastFaultOut,
	'Fast fault did not trip the beam');
	
	
//FFO remains faulted until local (FF) and FFO receieve fresh reset request, and faults
//are actually cleared

//Attempt to clear FFO fails because FF still faulted
fbFFO(i_xReset := TRUE); //Reset requested

fbFF(io_fbFFHWO := fbFFO, //FF faulted
	i_xOK := FALSE,
	i_xReset := FALSE);
	
fbFFO.EvaluateOutput(); //FFO eval called at end of cycle

AssertFalse(fbFFO.q_xFastFaultOut,
	'Fast fault output cleared while fault remains, very bad');
	
//Attempt to clear FF while fault remains fails
fbFFO(i_xReset := FALSE);
fbFFO(i_xReset := TRUE); //Reset requested

fbFF(io_fbFFHWO := fbFFO, //FF faulted
	i_xOK := FALSE,
	i_xReset := TRUE); //This reset should fail.
	
fbFFO.EvaluateOutput(); //FFO eval called at end of cycle

AssertFalse(fbFFO.q_xFastFaultOut,
	'Fast fault cleared while fault remains, very bad');
	
TEST_FINISHED();
END_METHOD

METHOD FFRegistration
VAR_INPUT
END_VAR
VAR
	fbFF	:	FB_FastFault;
	fbFFO	:	FB_HardwareFFOutput;
END_VAR
TEST('FFRegistration');

fbFF(io_fbFFHWO := fbFFO);

AssertEquals_STRING(fbFF.sPath, fbFFO.asList[fbFFO.nIndex-1],
	'FF registration with FFO did not succeed');

TEST_FINISHED();
END_METHOD

END_FUNCTION_BLOCK

// ---- pmps-lib/TestComponents/FB_Arbiter_Test.TcPOU
{attribute 'call_after_init'}
FUNCTION_BLOCK FB_Arbiter_Test EXTENDS TcUnit.FB_TestSuite
VAR_INPUT
END_VAR
VAR_OUTPUT
END_VAR
VAR
END_VAR

Arbitration();
RequestCheckRemoveBP();

METHOD Arbitration
VAR_INPUT
END_VAR
VAR
	fbArbiter	:	FB_Arbiter;
	
 	nAttReqID	:	UDINT	:= 1;
	stAttReqBP	:	ST_BeamParams := PMPS_GVL_BeamParams.cstFullBeam;
	
	nPPEReqID	:	UDINT	:= 2;
	stPPEReqBP	:	ST_BeamParams := PMPS_GVL_BeamParams.cstFullBeam;
	
	nEVReqID	:	UDINT	:= 3;
	stEVReqBP	:	ST_BeamParams := PMPS_GVL_BeamParams.cstFullBeam;
	
	nRateReqID	:	UDINT	:= 4;
	stRateReqBP	:	ST_BeamParams := PMPS_GVL_BeamParams.cstFullBeam;
	
	stArbitratedBP	:	ST_BeamParams;
	stExpectedBP	:	ST_BeamParams;
END_VAR
TEST('Arbitration');

//Initialize arbiter
fbArbiter.A_Init();

stAttReqBP.fAtt := 50;
stPPEReqBP.fPP_mJ := 1;
stEVReqBP.neVRange := 2#1111_1100_1111_1111;
stRateReqBP.nRate := 120;

//Load arbiter with beam parameter sets
AssertTrue(fbArbiter.AddRequest(nAttReqID, stAttReqBP),
					'Safest attenuation request failed to load');
					
//Load arbiter with beam parameter sets
AssertTrue(fbArbiter.AddRequest(nPPEReqID, stPPEReqBP),
					'Safest PPE request failed to load');
					
//Load arbiter with beam parameter sets
AssertTrue(fbArbiter.AddRequest(nEVReqID, stEVReqBP),
					'Safest stEVReqBP request failed to load');
					
//Load arbiter with beam parameter sets
AssertTrue(fbArbiter.AddRequest(nRateReqID, stRateReqBP),
					'Safest stEVReqBP request failed to load');

stExpectedBP.fAtt 	:= 	stAttReqBP.fAtt;
stExpectedBP.fPP_mJ	:=  stPPEReqBP.fPP_mJ;
stExpectedBP.neVRange := stEVReqBP.neVRange;
stExpectedBP.nRate := stRateReqBP.nRate;

stArbitratedBP := fbArbiter.GetArbitratedBP();

AssertFalse(F_DiffReqBeamParams(stExpectedBP, stArbitratedBP),
				'Arbitrated BP does not match expected.');

TEST_FINISHED();
END_METHOD

METHOD RequestCheckRemoveBP
VAR_INPUT
END_VAR
VAR
	fbArbiter	:	FB_Arbiter;
	
	nId	:	DWORD := 1;
	stReq	:	ST_BeamParams;
END_VAR
fbArbiter.A_Init();

TEST('RequestBP');
AssertTrue(fbArbiter.AddRequest(nId, stReq),
	'Request failed');

TEST_FINISHED();
	
TEST('DuplicateID');
AssertFalse(fbArbiter.AddRequest(nId, stReq),
	'Duplicate request accepted, not good.');

TEST_FINISHED();
	
TEST('CheckBP');
AssertTrue(fbArbiter.CheckRequest(nId),
	'Check failed');

TEST_FINISHED();	
	
TEST('IDDoesNotExist');
AssertFalse(fbArbiter.CheckRequest(nId+1),
	'Check returned true when ID does not exist');

TEST_FINISHED();
	
TEST('RemoveBP');
AssertTrue(fbArbiter.RemoveRequest(nId),
	'Remove failed');
AssertFalse(fbArbiter.CheckRequest(nId),
	'Remove did not remove request');
	
TEST_FINISHED();
END_METHOD

END_FUNCTION_BLOCK

// ---- pmps-lib/HelperFunctions/F_DiffReqBeamParams.TcPOU
(*Compares BeamParam1 to BeamParam2, if any parameters of BeamParam1 are different than BeamParam2
the result will be true *)
FUNCTION F_DiffReqBeamParams : BOOL
VAR_INPUT
	BeamParam1	:	ST_BeamParams;
	BeamParam2	:	ST_BeamParams;
END_VAR
VAR
	// Internal Attenuation OK boolean
	xAttOK: BOOL := FALSE;
	// Internal Per-pulse energy OK boolean
	xPPmjOK: BOOL := FALSE;
	// Internal photon energy OK boolean
	xEvOK: BOOL := FALSE;
	xRateOK: BOOL;
END_VAR

xAttOK := BeamParam1.fAtt <> BeamParam2.fAtt;
xPPmjOK := BeamParam1.fPP_mJ <> BeamParam2.fPP_mJ;
xEvOK := BeamParam1.neVRange <> BeamParam2.neVRange;
xRateOK	 := BeamParam1.nRate <> BeamParam2.nRate;


F_DiffReqBeamParams := xAttOK OR xPPmjOK OR xEvOK OR xRateOK;

END_FUNCTION

// ---- pmps-lib/MajorComponents/FB_UsualSuspects.TcPOU
//Used to register fast faults
FUNCTION_BLOCK FB_UsualSuspects
VAR_INPUT
END_VAR
VAR_OUTPUT
END_VAR
VAR
	asList	:	ARRAY[0..cMaxList] OF T_MaxString;
	nIndex	:	INT;
END_VAR
VAR CONSTANT
	cMaxList	:	INT := 99;
END_VAR

METHOD M_Register : BOOL
VAR_INPUT
	i_sFFName	:	STRING; //Fast fault FB variable name to register
END_VAR

VAR
END_VAR
IF THIS^.nIndex <= THIS^.cMaxList THEN
	THIS^.asList[MIN(THIS^.nIndex,THIS^.cMaxList)]:=i_sFFName;
	THIS^.nIndex := THIS^.nIndex + 1;
	M_Register := TRUE; //Add successful
ELSE
	M_Register := FALSE; //failed to add name to list
END_IF
END_METHOD

END_FUNCTION_BLOCK

// ---- pmps-lib/HelperFunctions/F_DiffBeamParamsRB.TcPOU
(*Compares BeamParam1 to BeamParam2, if any parameters of BeamParam1 are different than BeamParam2
the result will be true *)
FUNCTION F_DiffBeamParamsRB : BOOL
VAR_INPUT
	BeamParam1	:	ST_BeamParams;
	BeamParam2	:	ST_BeamParams;
END_VAR
VAR
	// Internal Attenuation OK boolean
	xAttOK: BOOL := FALSE;
	// Internal Per-pulse energy OK boolean
	xPPmjOK: BOOL := FALSE;
	// Internal photon energy OK boolean
	xEvOK: BOOL := FALSE;
	xRateOK: BOOL;
END_VAR

xAttOK := BeamParam1.fAtt <> BeamParam2.fAtt;
xPPmjOK := BeamParam1.fPP_mJ <> BeamParam2.fPP_mJ;
xEvOK := BeamParam1.reV <> BeamParam2.reV;
xRateOK	 := BeamParam1.nRate <> BeamParam2.nRate;


F_DiffBeamParamsRB := xAttOK OR xPPmjOK OR xEvOK OR xRateOK;

END_FUNCTION

// ---- pmps-lib/HelperFunctions/F_DifferentBeamParams.TcPOU
{attribute 'obsolete' := 'Use Req and Readback BP structs instead.'} 
(*DEPRECATED Compares BeamParam1 to BeamParam2, if any parameters of BeamParam1 are different than BeamParam2
the result will be true. *)
FUNCTION F_DifferentBeamParams : BOOL
VAR_INPUT
	BeamParam1	:	ST_BeamParams;
	BeamParam2	:	ST_BeamParams;
END_VAR
VAR
	// Internal Attenuation OK boolean
	xAttOK: BOOL := FALSE;
	// Internal Per-pulse energy OK boolean
	xPPmjOK: BOOL := FALSE;
	// Internal photon energy OK boolean
	xEvOK: BOOL := FALSE;
	xRateOK: BOOL;
END_VAR

xAttOK := BeamParam1.fAtt <> BeamParam2.fAtt;
xPPmjOK := BeamParam1.fPP_mJ <> BeamParam2.fPP_mJ;
xEvOK := BeamParam1.neVRange <> BeamParam2.neVRange;
xRateOK	 := BeamParam1.nRate <> BeamParam2.nRate;


F_DifferentBeamParams := xAttOK OR xPPmjOK OR xEvOK OR xRateOK;

END_FUNCTION

// ---- pmps-lib/MajorComponents/FB_BeamClassOutputs.TcPOU
(*
Sets the beam class assertion lines for a given beam class.
*)
FUNCTION_BLOCK FB_BeamClassOutputs
VAR_INPUT
	i_ArbiterBP	:	ST_BeamParams;
END_VAR
VAR_OUTPUT
END_VAR
VAR
	wBeamClass	:	BYTE;
	q_BC_ASSERTION_LINES	AT	%Q*	: ARRAY [1..16] OF	BOOL;
	InitCounter: INT;
	counter	:	INT;
END_VAR


//Beam Class
////////////////////////////////////
//0x0 = 0000 0000 0000 0000
//0x1 = 0000 0000 0000 0001
//0xF = 1111 1111 1111 1111

//Initialize BC lines to zero on every pass
FOR InitCounter := 1 TO 16 DO
	q_BC_ASSERTION_LINES[InitCounter] := FALSE;
END_FOR

//Set BC lines according to beam class
//A BC of 0x0 would pass over this loop, setting none of the lines high
// , as FOR loops check the initialized variable at the top to see if it's >
// than the "TO" variable.
FOR wBeamClass:=1 TO i_ArbiterBP.nBeamClass DO
	q_BC_ASSERTION_LINES[wBeamClass] := TRUE;
END_FOR

END_FUNCTION_BLOCK

// ---- pmps-lib/TestComponents/FB_BeamParamFanout_Test.TcPOU
{attribute 'call_after_init'}
FUNCTION_BLOCK FB_BeamParamFanout_Test EXTENDS TcUnit.FB_TestSuite
VAR_INPUT
END_VAR
VAR_OUTPUT
END_VAR
VAR

END_VAR

METHOD PRIVATE BPFanoutSafeguard
VAR_INPUT
END_VAR
VAR
	fbBPF	:	FB_BeamParamFanout;
END_VAR
TEST('Reset validity bool if interface invalid');
fbBPF.xTxPDO_state := 0; //OP
fbBPF();
AssertTrue(fbBPF.stBP.xValidToggle,
	'Does not start valid');
	
fbBPF.xTxPDO_state := 1; // Not op	
	
AssertFalse(fbBPF.stBP.xValidToggle,
	'Does not indicate invalid after IF goes non-op');
END_METHOD

END_FUNCTION_BLOCK

// ---- pmps-lib/TestComponents/FB_BPRequestor_Test.TcPOU
{attribute 'call_after_init'}
FUNCTION_BLOCK FB_BPRequestor_Test EXTENDS TcUnit.FB_TestSuite
VAR_INPUT
END_VAR
VAR_OUTPUT
END_VAR
VAR

END_VAR

METHOD PRIVATE BPRequestorSafeGuardFunctionality
VAR_INPUT
END_VAR
VAR
	fbBPR	:	FB_BPRequestor;
END_VAR
TEST('Reset Beam to Safe if Arbiter Faulted');
END_METHOD

END_FUNCTION_BLOCK

// ---- pmps-lib/TestComponents/FB_evRangeCalculator_Test.TcPOU
{attribute 'call_after_init'}
FUNCTION_BLOCK FB_evRangeCalculator_Test EXTENDS FB_TestSuite
VAR_INPUT
END_VAR
VAR_OUTPUT
END_VAR
VAR
END_VAR

BasicFunction();

METHOD BasicFunction
VAR_INPUT
END_VAR
VAR
	LastWord : WORD := 2#0000_0000_0000_0010;
END_VAR
TEST('CheckRanges');
//Upper limit equal
AssertTrue(
	F_eVRangeCalculator(300, 0) = 2#0000_0000_0000_0110,
	'Upper limit not inclusive');
//Lower limit equal
AssertTrue(
	F_eVRangeCalculator(300, 0) = 2#0000_0000_0000_0110,
	'Upper limit not inclusive');
//Mid range
AssertTrue(
	F_eVRangeCalculator(251, 0) = 2#0000_0000_0000_0010,
	'In range failed, whatever you did, it broke this really bad.');
//Out of range
AssertFalse(
	F_eVRangeCalculator(300.1, 0) = 2#0000_0000_0000_0010,
	'Out of range failed, whatever you did, it broke this really bad.');

TEST_FINISHED();

TEST('Negative eV failsafes');
//Negative eV
AssertTrue(
	F_eVRangeCalculator(-300, 0) = 16#FFFF,
	'Working with antimatter? Negative eV should failsafe to FFFF.');	

TEST_FINISHED();

TEST('Check hyst keeps');

AssertTrue(
	F_eVRangeCalculator(350, 2#0000_0000_0000_0010) = 2#0000_0000_0000_0110,
	'Moving up does not stick.');
	
AssertTrue(
	F_eVRangeCalculator(150, 2#0000_0000_0000_0010) = 2#0000_0000_0000_0011,
	'Moving down does not stick.');

TEST_FINISHED();

TEST('Check hyst drops');

AssertTrue(
	F_eVRangeCalculator(351, 2#0000_0000_0000_0010) = 2#0000_0000_0000_0100,
	'Moving up does not drop.');
	
AssertTrue(
	F_eVRangeCalculator(149, 2#0000_0000_0000_0010) = 2#0000_0000_0000_0001,
	'Moving down does not drop.');

TEST_FINISHED();

TEST_FINISHED_NAMED('FOO');
END_METHOD

END_FUNCTION_BLOCK

// ---- pmps-lib/TestComponents/FB_SolidAttenuator.TcPOU
FUNCTION_BLOCK FB_SolidAttenuator
VAR_INPUT
	i_rRequestedAttenuation	:	REAL;
END_VAR
VAR_OUTPUT
	q_xFault	:	BOOL;
	q_rCurrentAttenuation	:	REAL;
END_VAR
VAR_IN_OUT
	Arbiter	:	FB_Arbiter; //Higher level arbiter from which upstream attenuation can be requested
END_VAR
VAR
	stAttenuator	:	ST_BinarySolidAttenuator;
	nSearchStart: INT;
	nArrayLength: INT;
	axNewBladeStates	:	ARRAY [0..9]	OF	BOOL;
	nTryIndex: INT;
	rCurrentAccumulatedAttenuation: REAL;
	rTryFilter: REAL;
	rTryAttenuation: REAL;
	rRequestedAttenuation: REAL;
END_VAR



//

//Assuming the blades are ordered thickest to thinnest 
REPEAT
	rTryAttenuation := rCurrentAccumulatedAttenuation + stAttenuator.axBlades[nTryIndex].rThickness;
	IF rRequestedAttenuation >= rTryAttenuation THEN
		rCurrentAccumulatedAttenuation := rTryAttenuation;
		axNewBladeStates[nTryIndex] := TRUE;
	ELSE
		axNewBladeStates[nTryIndex] := FALSE;
	END_IF
UNTIL
	nTryIndex >= nArrayLength
END_REPEAT

END_FUNCTION_BLOCK

// ---- POUs/DatabaseComponents/FB_ExampleDeviceSM_DB.TcPOU
(* This version of the block is self contained. Minimizes wiring.*)
FUNCTION_BLOCK FB_ExampleDeviceSM_DB
VAR_INPUT
	cBase: UDINT;
	iDBID:UDINT;
	sDBNetId: STRING;
	sDeviceID: STRING;
END_VAR
VAR_OUTPUT
END_VAR
VAR_IN_OUT
	fbArbiter : FB_Arbiter;
	fbFastFaultOutput	:	FB_HardwareFFOutput;
END_VAR
VAR
	stDevice	:	ST_Device;
	fbGovernor	:	FB_LinearGovernor;
	mcPower	:	MC_Power;
	mcStop: MC_Stop;
	mcAbsolute	:	MC_MoveAbsolute;
	fbBPTM	:	BeamParameterTransitionManager;
	xStartMove: BOOL;
	
	stCheckState: ST_DeviceState;
	stTargetState	:	ST_DeviceState; //Target device state
	fbDBClient:FB_MySQL_Client;
	bInitReady: BOOL :=FALSE;
	//aStateTable : ARRAY[1..MAX_DEVICE_STATES] OF ST_DeviceStateTable;

END_VAR
VAR PERSISTENT
	nLastActiveState	:	UDINT;
END_VAR

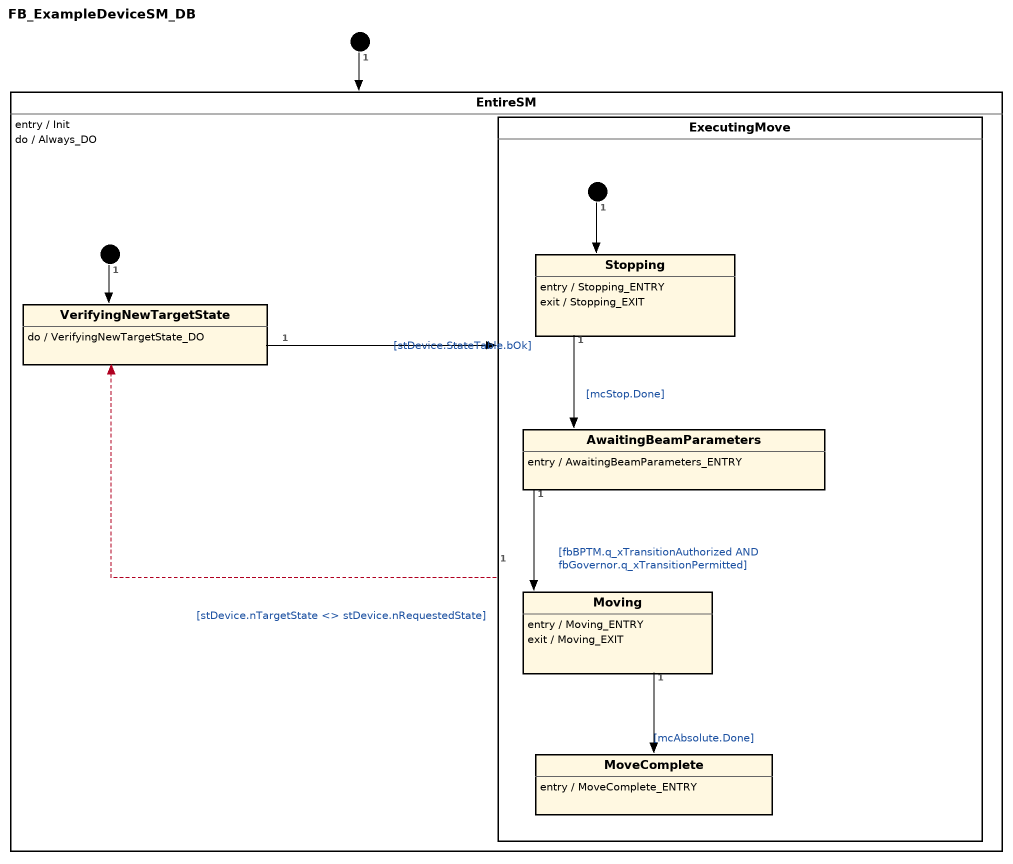
STATECHART FB_ExampleDeviceSM_DB  // abortable
    START StartState3
    COMPOSITE STATE EntireSM
        entry / Init
        do / Always_DO
        START StartState1
        COMPOSITE STATE ExecutingMove
            START StartState2
            STATE Stopping
                entry / Stopping_ENTRY
                exit / Stopping_EXIT
            STATE AwaitingBeamParameters
                entry / AwaitingBeamParameters_ENTRY
            STATE Moving
                entry / Moving_ENTRY
                exit / Moving_EXIT
            STATE MoveComplete
                entry / MoveComplete_ENTRY
            StartState2 -> Stopping  // priority 1, on completion
            Stopping -> AwaitingBeamParameters [mcStop.Done] // priority 1, rising edge
            AwaitingBeamParameters -> Moving [fbBPTM.q_xTransitionAuthorized AND fbGovernor.q_xTransitionPermitted] // priority 1, rising edge
            Moving -> MoveComplete [mcAbsolute.Done] // priority 1, rising edge
        END_STATE
        STATE VerifyingNewTargetState
            do / VerifyingNewTargetState_DO
        StartState1 -> VerifyingNewTargetState  // priority 1, on completion
        ExecutingMove -> VerifyingNewTargetState [stDevice.nTargetState <> stDevice.nRequestedState] // priority 1, exception, rising edge
        VerifyingNewTargetState -> ExecutingMove [stDevice.StateTable.bOk] // priority 1
    END_STATE
    StartState3 -> EntireSM  // priority 1, on completion
END_STATECHART

ACTION Always_DO:
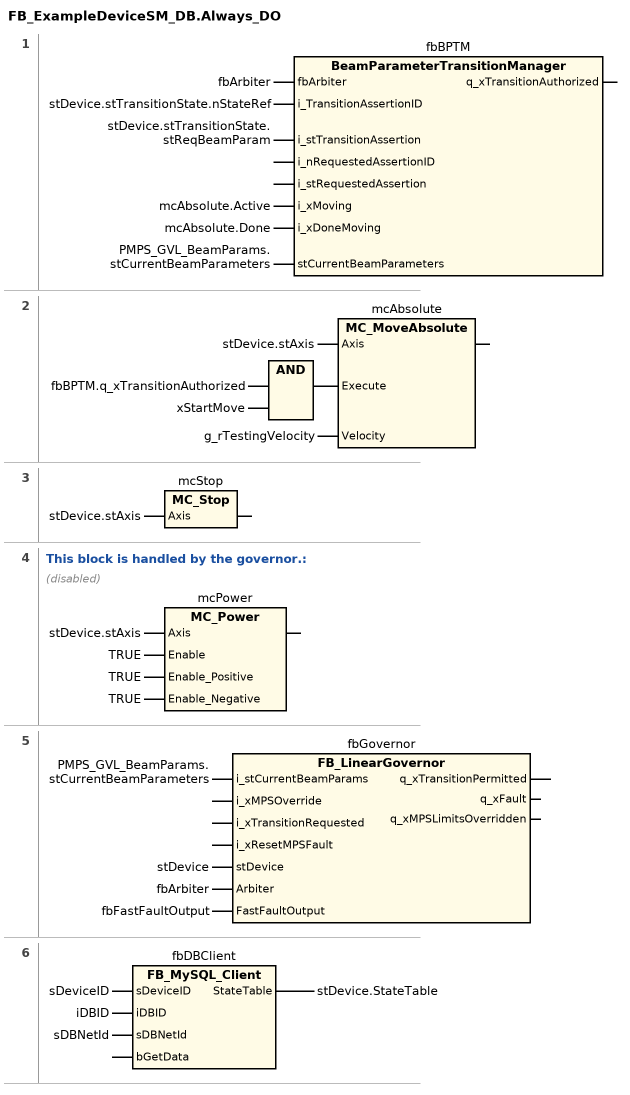
// NETWORK 1
fbBPTM(
    fbArbiter := fbArbiter,
    i_TransitionAssertionID := stDevice.stTransitionState.nStateRef,
    i_stTransitionAssertion := stDevice.stTransitionState.stReqBeamParam,
    i_xMoving := mcAbsolute.Active,
    i_xDoneMoving := mcAbsolute.Done,
    stCurrentBeamParameters := PMPS_GVL_BeamParams.stCurrentBeamParameters); // BeamParameterTransitionManager

// NETWORK 2
mcAbsolute(
    Axis := stDevice.stAxis,
    Execute := fbBPTM.q_xTransitionAuthorized AND xStartMove,
    Velocity := g_rTestingVelocity); // MC_MoveAbsolute

// NETWORK 3
mcStop(Axis := stDevice.stAxis); // MC_Stop

// NETWORK 4 (disabled)
// label: This block is handled by the governor.
// mcPower(Axis := stDevice.stAxis, Enable := TRUE, Enable_Positive := TRUE, Enable_Negative := TRUE); // MC_Power

// NETWORK 5
fbGovernor(
    i_stCurrentBeamParams := PMPS_GVL_BeamParams.stCurrentBeamParameters,
    stDevice := stDevice,
    Arbiter := fbArbiter,
    FastFaultOutput := fbFastFaultOutput); // FB_LinearGovernor

// NETWORK 6
fbDBClient(sDeviceID := sDeviceID, iDBID := iDBID, sDBNetId := sDBNetId); // FB_MySQL_Client
stDevice.StateTable := fbDBClient.StateTable;
END_ACTION

ACTION AwaitingBeamParameters_ENTRY:
fbBPTM.i_stRequestedAssertion := stTargetState.stReqBeamParam;
fbBPTM.i_nRequestedAssertionID := stTargetState.nStateRef;

//Tell the governor that we're trying to move.
fbGovernor.i_xTransitionRequested := TRUE;
END_ACTION

ACTION Init:
	
//Safe State
stDevice.nSafeState := cBase;
stDevice.nTransitionState := cBase+100;

//Initialize the State Table
stDevice.StateTable.A_Reset();
//Device State Table Instantiation
F_SetStateParams(
	nStateRef := stDevice.nSafeState,
	rPosition := 0,
	rTolerance := 10,
	stBeamParams := PMPS_GVL_BeamParams.cstFullBeam,
	Table := stDevice.StateTable
);
//Connect to DB and get state table data
fbDBClient.bGetData:= TRUE;//fbMySQL.nState:=400; 

stDevice.StateTable.A_Lookup(
		key := stDevice.nTransitionState,
		getValue => stDevice.stTransitionState
);
	
//Need an initialization routine for setting the active state
//Check if the device is at the last known state
//If the device is within the state boundaries, it's considered to be in that state
stDevice.StateTable.A_Lookup(key:= nLastActiveState);
IF stDevice.StateTable.bOk THEN
	stCheckState := stDevice.StateTable.getValue;
ELSE
	stCheckState := stDevice.stTransitionState; //This needs to be safer <TODO>
END_IF

IF stDevice.stAxis.NcToPlc.ActPos <= stCheckstate.rPosition + stCheckState.rTolerance AND
	stDevice.stAxis.NcToPlc.ActPos >= stCheckState.rPosition - stCheckState.rTolerance THEN
	stDevice.nActiveState := nLastActiveState;
ELSE
	stDevice.nActiveState := stDevice.nTransitionState;
END_IF

//Simulation Hardware Limit Switches
stDevice.i_xHiLim := TRUE;
stDevice.i_xLoLim := TRUE;
END_ACTION

ACTION Initialize:

END_ACTION

ACTION MoveComplete_ENTRY:
//Clear transition request
fbGovernor.i_xTransitionRequested := FALSE;
//Latch active state
stDevice.nActiveState := stDevice.nTargetState;
nLastActiveState := stDevice.nActiveState;
END_ACTION

ACTION Moving_ENTRY:
xStartMove := TRUE;
mcAbsolute.Position := stTargetState.rPosition;
END_ACTION

ACTION Moving_EXIT:
xStartMove := FALSE;
END_ACTION

ACTION NewMove_ENTRY:

END_ACTION

ACTION Stopping_ENTRY:
mcStop.Execute := TRUE;
END_ACTION

ACTION Stopping_EXIT:
mcStop.Execute := FALSE;
END_ACTION

ACTION VerifyingNewTargetState_DO:
stDevice.StateTable.A_Lookup(
	key := stDevice.nRequestedState
);

IF stDevice.StateTable.bOk THEN
	stTargetState := stDevice.StateTable.getValue;
	stDevice.nTargetState := stDevice.nRequestedState;
ELSE
	; //log ignored state/ generate an error? <TODO>
END_IF
END_ACTION

END_FUNCTION_BLOCK

// ---- POUs/DatabaseComponents/FB_MySQL_Client.TcPOU
FUNCTION_BLOCK FB_MySQL_Client
VAR_INPUT
	sDeviceID: STRING;
	iDBID:UDINT;
	sDBNetId: STRING ;
	bGetData:BOOL;
END_VAR
VAR_OUTPUT
	StateTable : FB_LinearDeviceStateTable;
END_VAR
VAR CONSTANT
	sSQLCommand :STRING:='SELECT * FROM device_states  WHERE device_id =';
END_VAR
VAR
	nState: INT:=0; // used as a start signal
	nRecordCount: UDINT:=MAX_DEVICE_STATES;
	aDeviceStateTable : ARRAY[1..MAX_DEVICE_STATES] OF ST_DeviceStateTable;
	fbMySQLDB:  FB_SQLDatabase(sNetId := '', tTimeout:=T#5S);
	fbSQLCmd:  FB_SQLCommand(sNetId := '', tTimeout:=T#5S);
	fbSQLResult: FB_SQLResult(sNetId := '', tTimeout:=T#5S);
	sSQLCmd :STRING;
	ipResultEvent : Tc3_Eventlogger.I_TcResultEvent;
	
	
END_VAR


IF (bGetData) THEN
	bGetData:= FALSE;
	nState := 100;
END_IF

CASE nState OF
	0:
100:// Initialize Database function blocks
	fbMySQLDB.sNetID := sDBNetId;
	fbSQLCmd.sNetID := sDBNetId;
	fbSQLResult.sNetID := sDBNetId; 
	IF fbMySQLDB.Connect(iDBID) THEN
		IF fbMySQLDB.bError THEN
			nState := 9000+nState; 
		ELSE
			nState := nState+1; 
		END_IF
	END_IF
 
101:	
	 IF(fbMySQLDB.bConnected ) THEN
		fbMySQLDB.CreateCmd(pSQLCommand := ADR(fbSQLCmd));
		IF fbMySQLDB.bError THEN
			nState := 9000+nState; 
		ELSE
			nState := 1+nState; 
		END_IF
	 END_IF
102:	 
  (*Execute SQL Comnmand*)
	//sSQLCmd :=sSQLCommand;
	sSQLCmd := CONCAT(sSQLCommand, sDeviceID) ;		
   IF fbSQLCmd.ExecuteDataReturn(pSQLCmd:=ADR(sSQLCmd),cbSQLCmd:=SIZEOF(sSQLCmd),pSQLDBResult:=ADR(fbSQLResult)) THEN
   	IF( fbSQLCmd.bError) THEN
	    nState := 9000+nState; 
    ELSE
        nState := 1+nState; 
		MEMSET(ADR(aDeviceStateTable),0,SIZEOF(aDeviceStateTable));

    END_IF
  END_IF
 
103: 
	(*Read data FROM the database*)
  IF (fbSQLResult.Read(nStartIndex:=0, nRecordCount:=nRecordCount,pData:=ADR(aDeviceStateTable),cbData:=SIZEOF(aDeviceStateTable),bWithVerifying:=TRUE,bDataRelease:=TRUE) )THEN
	 ipResultEvent := fbSQLResult.ipTcResultEvent;
	IF fbSQLResult.bError THEN
         nState := 9000+nState; 
    ELSE
        nState := 500;// 1+nState; 
    END_IF
END_IF	

500:
	//Device State Table Instantiation
	IF F_DB_To_hTable( aStatesParamsTable:= aDeviceStateTable, nRecordCount:=nRecordCount, Table := StateTable)THEN
         nState := 9000+nState; 
    ELSE
        nState :=800;// 1+nState; 
    END_IF



600: //Reload DATA
//Reset all hash table entries
// re instantiate device state table	
	;
9500:
800: //Release and Disconnect
	
	IF (fbSQLResult.Release() AND fbMySQLDB.Disconnect()) THEN
		nState:=-1;
		ELSE
			 nState := 9000+nState; 
	END_IF


		;
END_CASE

END_FUNCTION_BLOCK

// ---- POUs/DatabaseComponents/F_DB_To_hTable.TcPOU
FUNCTION F_DB_To_hTable : BOOL
VAR_INPUT
	aStatesParamsTable : ARRAY[1..MAX_DEVICE_STATES] OF ST_DeviceStateTable;
	nRecordCount: UDINT;
END_VAR
VAR_IN_OUT
	Table	:	FB_LinearDeviceStateTable;
END_VAR
VAR
	stDeviceState	:	ST_DeviceState;
	iRow : UDINT:=1;
END_VAR

Table.A_Reset();
//Device State Table Instantiation
(*F_SetStateParams(
	nStateRef := 0,
	rPosition := 0,
	rTolerance := 0,
	stBeamParams := PMPS_GVL_BeamParams.cstFullBeam,
	Table := Table
);
*)
IF (nRecordCount>0) THEN
	FOR iRow:=1 TO nRecordCount BY 1 DO
	stDeviceState.nStateRef := DINT_TO_UDINT(aStatesParamsTable[iRow].iStateID);
	stDeviceState.rPosition := aStatesParamsTable[iRow].rTargetPosition;
	stDeviceState.rTolerance := aStatesParamsTable[iRow].rTolerance;  
	stDeviceState.stReqBeamParam.fAtt := aStatesParamsTable[iRow].rTransmission;
	stDeviceState.stReqBeamParam.fPP_mJ := (aStatesParamsTable[iRow].rPerPulseEnergy);
	stDeviceState.stReqBeamParam.nRate := DINT_TO_UDINT(aStatesParamsTable[iRow].iPulseRate);
	stDeviceState.stReqBeamParam.nBeamClass := DINT_TO_BYTE(aStatesParamsTable[iRow].iBeamClass);
//	stDeviceState.stReqBeamParam.fUpper_eV := (aStatesParamsTable[iRow].rUpper_eV);
//	stDeviceState.stReqBeamParam.fLower_eV := (aStatesParamsTable[iRow].rLower_eV);
	stDeviceState.stReqBeamParam.reV := aStatesParamsTable[iRow].rPhotonEnergy;
	//stDeviceState.stReqBeamParam.neVRange := (aStatesParamsTable[iRow].rLower_eV);
	Table.A_Add(
		key := stDeviceState.nStateRef,
		putValue := stDeviceState
	);
END_FOR;
END_IF

Table.A_Count();
F_DB_To_hTable := Table.bOk;

END_FUNCTION

// ---- POUs/DeviceImplementationEx1/FB_ExampleDeviceSM.TcPOU

FUNCTION_BLOCK FB_ExampleDeviceSM
VAR_INPUT
	i_xMoveStarted	:	BOOL; //Connect to moving flag
	i_xMoveDone	:	BOOL; //Connect to move done flag
	i_xBeamReady	:	BOOL; //Connect to transitioneer
	i_xStopDone	:	BOOL; //Connect to MC_Stop.Done
END_VAR
VAR_OUTPUT
	q_xStartMove	:	BOOL; //Connect to MC_Absolute.Execute
	q_xStop			:	BOOL; //Connect to MC_Stop.Execute
	q_rTargetPosition	:	REAL; //Connect to MC_Absolute.Position
	q_stRequiredBeamParametersID	:	UDINT;
	q_stRequiredBeamParameters	:	ST_BeamParams; //Connect to BeamParameterTransitionManager
END_VAR
VAR_IN_OUT
	stDevice	:	ST_Device;
END_VAR
VAR
	nTargetState	:	INT;
	
	xNewReq	:	BOOL; //Set true when new target request present
	
END_VAR

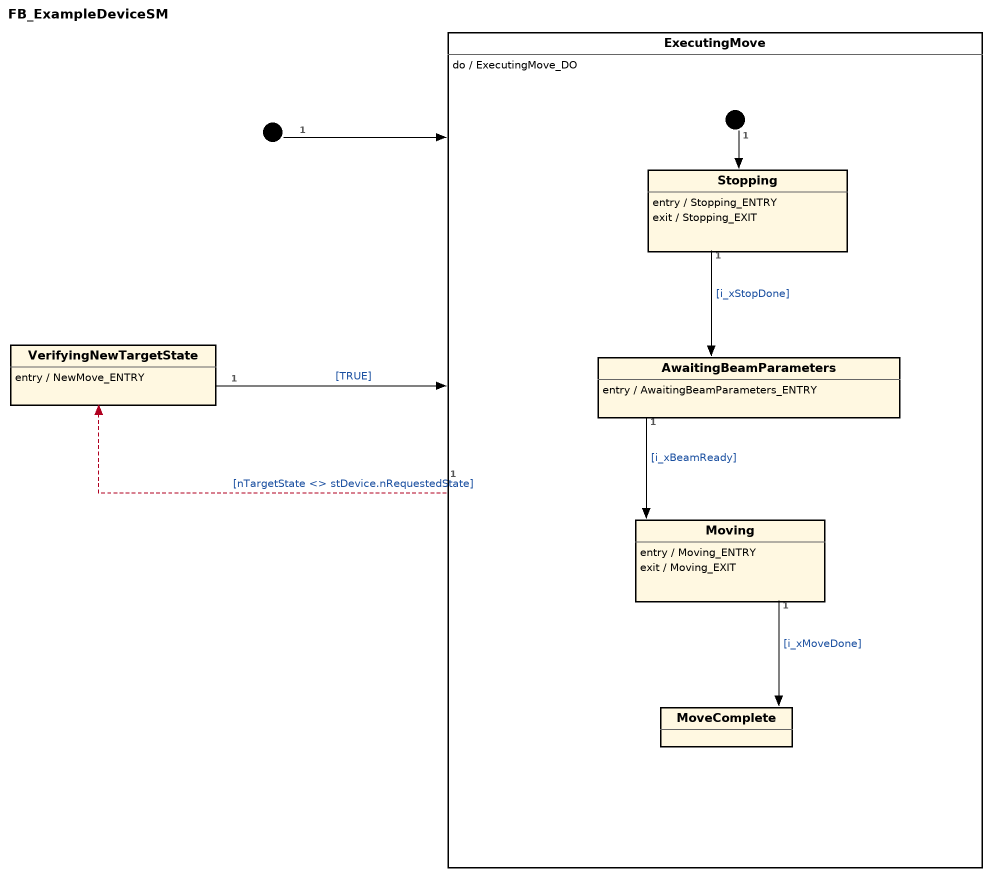
STATECHART FB_ExampleDeviceSM  // abortable
    START StartState1
    COMPOSITE STATE ExecutingMove
        do / ExecutingMove_DO
        START StartState2
        STATE Stopping
            entry / Stopping_ENTRY
            exit / Stopping_EXIT
        STATE AwaitingBeamParameters
            entry / AwaitingBeamParameters_ENTRY
        STATE Moving
            entry / Moving_ENTRY
            exit / Moving_EXIT
        STATE MoveComplete
        StartState2 -> Stopping  // priority 1, on completion
        Stopping -> AwaitingBeamParameters [i_xStopDone] // priority 1, rising edge
        AwaitingBeamParameters -> Moving [i_xBeamReady] // priority 1, rising edge
        Moving -> MoveComplete [i_xMoveDone] // priority 1, rising edge
    END_STATE
    STATE VerifyingNewTargetState
        entry / NewMove_ENTRY
    StartState1 -> ExecutingMove  // priority 1, on completion
    ExecutingMove -> VerifyingNewTargetState [nTargetState <> stDevice.nRequestedState] // priority 1, exception, rising edge
    VerifyingNewTargetState -> ExecutingMove [TRUE] // priority 1
END_STATECHART

ACTION AwaitingBeamParameters_ENTRY:
q_stRequiredBeamParameters := stDevice.astStates[nTargetState].stReqBeamParam;
q_stRequiredBeamParametersID := stDevice.astStates[nTargetState].nStateRef;
END_ACTION

ACTION ExecutingMove_DO:

END_ACTION

ACTION Moving_ENTRY:
q_xStartMove := TRUE;
q_rTargetPosition := stDevice.astStates[nTargetState].rPosition;
END_ACTION

ACTION Moving_EXIT:
q_xStartMove := FALSE;
END_ACTION

ACTION NewMove_ENTRY:

IF stDevice.nRequestedState <= PMPS_GVL_BeamParams.cnMaxStateArrayLen AND
	stDevice.nRequestedState >= 1 THEN
	nTargetState := stDevice.nRequestedState;
END_IF
END_ACTION

ACTION Stopping_ENTRY:
q_xStop	:= TRUE;
END_ACTION

ACTION Stopping_EXIT:
q_xStop := FALSE;
END_ACTION

END_FUNCTION_BLOCK

// ---- GlobalTextList.TcGTLO
TEXTLIST GlobalTextList
  788 = '%1.4f'
  333 = '%16b'
  646 = '%2b'
  108 = '%3.2f'
  476 = '%b'
  632 = '%d'
  993 = '%f'
  697 = '%x'
  441 = 'Actuator Position'
  511 = 'Arbiter Assertions'
  482 = 'Arbiter Stats'
  300 = 'Assertion Count'
  843 = 'Assertion ID'
  826 = 'Assertion Pool'
  68 = 'Assertion Pool State'
  766 = 'Assertion Pool Stats'
  708 = 'Att'
  276 = 'Attenuation'
  637 = 'cBase + 1 to move to a non-zero state. cBase is always "safe" state.'
  386 = 'cBase: %d'
  941 = 'Clear'
  20 = 'Clear Fault'
  52 = 'Clear Faults'
  983 = 'Current eV Range'
  992 = 'Current eV: %f'
  957 = 'eV'
  660 = 'Fast Fault'
  796 = 'Free Slots'
  42 = 'Governor Fault'
  688 = 'Governor Overridden'
  100 = 'GroupBox'
  284 = 'Imager'
  447 = 'Imager 1'
  330 = 'Imager 2'
  870 = 'lock'
  217 = 'Lower eV'
  585 = 'Machine Parameters'
  419 = 'MPS Override'
  520 = 'MPS Override Mode'
  967 = 'MPS Upper Limit'
  682 = 'NA'
  950 = 'nStateRef'
  434 = 'Override MPS'
  934 = 'Photon Energy'
  512 = 'Photon Energy Adjustment'
  514 = 'Photon Energy Ranges: %16b'
  605 = 'Photon Energy Ranges: %b'
  124 = 'Photon Energy Ranges: %d'
  465 = 'Photon Energy: %3.2f'
  667 = 'pNext'
  410 = 'PPE'
  650 = 'Pulse Energy'
  479 = 'Rate'
  710 = 'Requested eV Range'
  326 = 'rPosition'
  509 = 'rTolerance'
  978 = 'Select State'
  140 = 'sParentDevice'
  915 = 'sStateName'
  29 = 'State 1'
  57 = 'State 2'
  955 = 'State 3'
  290 = 'State Control'
  553 = 'stReqBeamParam'
  13 = 'Upper eV'
  396 = 'value'
END_TEXTLIST

// ---- VISUs/ArbiterStats.TcVIS
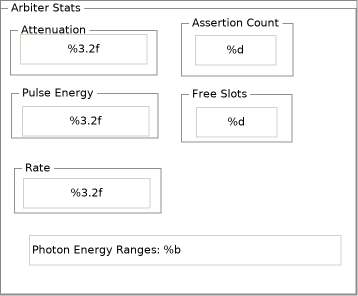
VISUALIZATION ArbiterStats  // 358x296
VAR_IN_OUT
	fbArbiter	:	FB_Arbiter;
END_VAR
    GroupBox (0,0 356x294), "Arbiter Stats"
        GroupBox (10,22 147x53), "Attenuation"
            Textfield (10,12 127x30), "%3.2f", text variable: fbArbiter.q_stBeamParams.fAtt
        GroupBox (11,85 147x53), "Pulse Energy"
            Textfield (11,21 127x30), "%3.2f", text variable: fbArbiter.q_stBeamParams.fPP_mJ
        GroupBox (14,160 147x53), "Rate"
            Textfield (9,18 127x30), "%3.2f", text variable: fbArbiter.stOutputBP.nRate
        GroupBox (181,15 112x61), "Assertion Count"
            Textfield (14,20 81x30), "%d", text variable: fbArbiter.fbBPAssertionPool.hTable.nCount
        GroupBox (181,86 111x56), "Free Slots"
            Textfield (15,21 81x30), "%d", text variable: fbArbiter.fbBPAssertionPool.hTable.nFree
        Textfield (29,235 312x30), "Photon Energy Ranges: %b", text variable: fbArbiter.q_stBeamParams.neVReqRange
END_VISUALIZATION

// ---- VISUs/BeamParameterStats.TcVIS
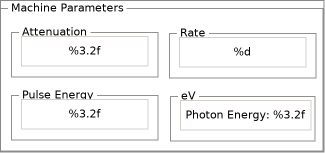
VISUALIZATION BeamParameterStats  // 325x153
VAR_IN_OUT
	BP	:	ST_BeamParams;
END_VAR
    GroupBox (0,0 323x151), "Machine Parameters"
        GroupBox (11,24 147x53), "Attenuation"
            Textfield (10,12 127x30), "%3.2f", text variable: BP.fAtt
        GroupBox (11,87 147x53), "Pulse Energy"
            Textfield (10,12 127x30), "%3.2f", text variable: BP.fPP_mJ
        GroupBox (169,25 147x53), "Rate"
            Textfield (10,12 127x30), "%d", text variable: BP.nRate
        GroupBox (170,88 145x53), "eV"
            Textfield (10,12 131x30), "Photon Energy: %3.2f", text variable: BP.reV
END_VISUALIZATION

// ---- VISUs/FastFaultGUI.TcVIS
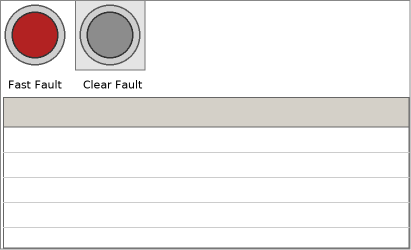
VISUALIZATION FastFaultGUI  // 411x250
VAR_IN_OUT
	FastFault	:	FB_HardwareFFOutput;
END_VAR
    Lamp1 (0,0 70x70), variable: NOT FastFault.q_xFastFaultOut, style: Lamp-Lamp1-Red
    Label (5,70 59x30), "Fast Fault"
    PushSwitch (75,0 70x70), variable: FastFault.i_xReset, behaviour: TAP, style: Switch-PushSwitch-Gray
    Label (80,70 59x30), "Clear Fault"
    Table (3,97 406x151), data array: FastFault.asList
        p3854506369: FastFault.asList[INDEX]
END_VISUALIZATION

// ---- VISUs/ImagerGUI.TcVIS
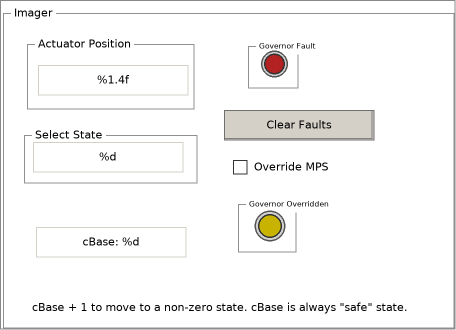
VISUALIZATION ImagerGUI  // 456x330
VAR_IN_OUT
	fbDevice	:	FB_ExampleDeviceSM_All;
END_VAR
    GroupBox (3,5 451x323), "Imager"
        Button (221,105 150x30), "Clear Faults"
            tap fbDevice.stDevice.xClearFaults
        Checkbox (228,147 150x30), "Override MPS", variable: fbDevice.stDevice.xOverrideMPSLimits
        GroupBox (245,33 50x50), "Governor Fault"
            Lamp1 (11,10 31x32), variable: fbDevice.stDevice.xGovernorFault, style: Lamp-Lamp1-Red
        GroupBox (235,191 58x56), "Governor Overridden"
            Lamp1 (14,10 36x40), variable: fbDevice.stDevice.xGovernorOverridden, style: Lamp-Lamp1-Yellow
        GroupBox (24,31 167x73), "Actuator Position"
            Textfield (11,29 150x30), "%1.4f", text variable: fbDevice.stDevice.stAxis.NcToPlc.ActPos
        GroupBox (21,122 173x56), "Select State"
            Textfield (9,15 150x30), "%d", tooltip "cBase + 1 to move to a non-zero state. cBase is always "safe" state.", text variable: fbDevice.stDevice.nRequestedState
                OnMouseDown: write the text variable via Default
        Label (33,293 368x19), "cBase + 1 to move to a non-zero state. cBase is always "safe" state."
        Textfield (33,222 150x30), "cBase: %d", tooltip "cBase + 1 to move to a non-zero state. cBase is always "safe" state.", text variable: fbDevice.cBase
            OnMouseDown: write the text variable via Default
END_VISUALIZATION

// ---- VISUs/PhotonEnergyWatcher.TcVIS
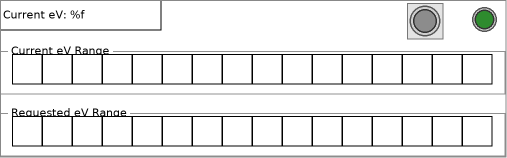
VISUALIZATION PhotonEnergyWatcher  // 507x158
VAR_IN_OUT
	Watcher	:	FB_PhotonEnergyWatcher;
END_VAR
    GroupBox (0,43 505x51), "Current eV Range"
        Frame (12,11 485x32)
            shows WordBitDisplay(nVal := Watcher.i_stCurrentBeamParams.neVRange)
    Rectangle (0,0 161x30), "Current eV: %f", text variable: Watcher.i_stCurrentBeamParams.reV
    GroupBox (0,105 505x51), "Requested eV Range"
        Frame (12,11 485x32)
            shows WordBitDisplay(nVal := Watcher.i_stRequestedBeamParams.neVRange)
    Lamp1 (470,2 29x35), variable: Watcher.fbFF.bsFF.Q1, style: Lamp-Lamp1-Green
    PushSwitch (407,1 36x40), variable: Watcher.i_xReset, behaviour: TAP, style: Switch-PushSwitch-Gray
END_VISUALIZATION

